LIN {X 0,Y 573.005,Z 611.639,A -85,B 0,C 180,E1 -2254.218,E2 -2254.218} C_VEL
LIN {X 0,Y 573.014,Z 607.193,A -85,B 0,C 180,E1 -2255.982,E2 -2255.982} C_VEL
LIN {X 0,Y 573.04,Z 602.476,A -85,B 0,C 180,E1 -2257.397,E2 -2257.397} C_VEL
LIN {X 0,Y 573.091,Z 594.867,A -85,B 0,C 180,E1 -2259.171,E2 -2259.171} C_VEL
LIN {X 0,Y 573.165,Z 587.276,A -85,B 0,C 180,E1 -2260.596,E2 -2260.596} C_VEL
LIN {X 0,Y 573.302,Z 578.228,A -85,B 0,C 180,E1 -2262.026,E2 -2262.026} C_VEL
LIN {X 0,Y 573.441,Z 567.442,A -85,B 0,C 180,E1 -2263.463,E2 -2263.463} C_VEL
LIN {X 0,Y 573.682,Z 556.314,A -85,B 0,C 180,E1 -2264.723,E2 -2264.723} C_VEL
LIN {X 0,Y 573.877,Z 544.168,A -85,B 0,C 180,E1 -2265.901,E2 -2265.901} C_VEL
LIN {X 0,Y 574.13,Z 530.904,A -85,B 0,C 180,E1 -2266.991,E2 -2266.991} C_VEL
LIN {X 0,Y 574.389,Z 517.891,A -85,B 0,C 180,E1 -2267.901,E2 -2267.901} C_VEL
LIN {X 0,Y 574.662,Z 504.072,A -85,B 0,C 180,E1 -2268.723,E2 -2268.723} C_VEL
LIN {X 0,Y 574.932,Z 489.306,A -85,B 0,C 180,E1 -2269.448,E2 -2269.448} C_VEL
LIN {X 0,Y 575.133,Z 474.014,A -85,B 0,C 180,E1 -2270.052,E2 -2270.052} C_VEL
LIN {X 0,Y 575.364,Z 457.285,A -85,B 0,C 180,E1 -2270.557,E2 -2270.557} C_VEL
LIN {X 0,Y 575.514,Z 441.109,A -85,B 0,C 180,E1 -2270.902,E2 -2270.902} C_VEL
LIN {X 0,Y 576.207,Z 242.353,A -85,B 0,C 180,E1 -2273.515,E2 -2273.515} C_VEL
LIN {X 0,Y 575.024,Z 234.784,A -85,B 0,C 180,E1 -2273.687,E2 -2273.687} C_VEL
LIN {X 0,Y 575.523,Z 201.562,A -85,B 0,C 180,E1 -2276.564,E2 -2276.564} C_VEL
LIN {X 0,Y 575.358,Z 193.757,A -85,B 0,C 180,E1 -2277.259,E2 -2277.259} C_VEL
LIN {X 0,Y 573.235,Z 186.394,A -85,B 0,C 180,E1 -2278.026,E2 -2278.026} C_VEL
LIN {X 0,Y 573.213,Z 186.396,A -85,B 0,C 180,E1 -2280.88,E2 -2280.88} C_VEL
LIN {X 0,Y 573.245,Z 186.393,A -85,B 0,C 180,E1 -2283.522,E2 -2283.522} C_VEL
LIN {X 0,Y 573.196,Z 186.394,A -85,B 0,C 180,E1 -2286.049,E2 -2286.049} C_VEL
LIN {X 0,Y 573.225,Z 186.392,A -85,B 0,C 180,E1 -2288.699,E2 -2288.699} C_VEL
LIN {X 0,Y 573.209,Z 186.396,A -85,B 0,C 180,E1 -2291.455,E2 -2291.455} C_VEL
LIN {X 0,Y 573.208,Z 186.391,A -85,B 0,C 180,E1 -2294.332,E2 -2294.332} C_VEL
LIN {X 0,Y 573.222,Z 186.395,A -85,B 0,C 180,E1 -2297.356,E2 -2297.356} C_VEL
LIN {X 0,Y 573.223,Z 186.389,A -85,B 0,C 180,E1 -2300.391,E2 -2300.391} C_VEL
LIN {X 0,Y 573.227,Z 186.396,A -85,B 0,C 180,E1 -2303.076,E2 -2303.076} C_VEL
LIN {X 0,Y 573.242,Z 186.388,A -85,B 0,C 180,E1 -2305.67,E2 -2305.67} C_VEL
LIN {X 0,Y 573.22,Z 186.387,A -85,B 0,C 180,E1 -2308.184,E2 -2308.184} C_VEL
LIN {X 0,Y 573.236,Z 186.392,A -85,B 0,C 180,E1 -2310.633,E2 -2310.633} C_VEL
LIN {X 0,Y 573.227,Z 186.394,A -85,B 0,C 180,E1 -2313.023,E2 -2313.023} C_VEL
LIN {X 0,Y 573.242,Z 186.39,A -85,B 0,C 180,E1 -2315.365,E2 -2315.365} C_VEL
LIN {X 0,Y 573.233,Z 186.388,A -85,B 0,C 180,E1 -2317.662,E2 -2317.662} C_VEL
LIN {X 0,Y 573.245,Z 186.39,A -85,B 0,C 180,E1 -2320.727,E2 -2320.727} C_VEL
LIN {X 0,Y 573.225,Z 186.389,A -85,B 0,C 180,E1 -2323.621,E2 -2323.621} C_VEL
LIN {X 0,Y 573.211,Z 186.394,A -85,B 0,C 180,E1 -2326.529,E2 -2326.529} C_VEL
LIN {X 0,Y 573.262,Z 186.384,A -85,B 0,C 180,E1 -2329.404,E2 -2329.404} C_VEL
LIN {X 0,Y 573.256,Z 186.387,A -85,B 0,C 180,E1 -2332.25,E2 -2332.25} C_VEL
LIN {X 0,Y 573.283,Z 186.381,A -85,B 0,C 180,E1 -2335.077,E2 -2335.077} C_VEL
LIN {X 0,Y 573.267,Z 186.38,A -85,B 0,C 180,E1 -2337.893,E2 -2337.893} C_VEL
LIN {X 0,Y 573.316,Z 186.387,A -85,B 0,C 180,E1 -2340.703,E2 -2340.703} C_VEL
LIN {X 0,Y 573.206,Z 186.389,A -85,B 0,C 180,E1 -2343.515,E2 -2343.515} C_VEL
LIN {X 0,Y 573.257,Z 186.382,A -85,B 0,C 180,E1 -2345.629,E2 -2345.629} C_VEL
LIN {X 0,Y 573.275,Z 186.39,A -85,B 0,C 180,E1 -2348.46,E2 -2348.46} C_VEL
LIN {X 0,Y 573.265,Z 186.381,A -85,B 0,C 180,E1 -2351.313,E2 -2351.313} C_VEL
LIN {X 0,Y 573.247,Z 186.393,A -85,B 0,C 180,E1 -2354.426,E2 -2354.426} C_VEL
LIN {X 0,Y 573.269,Z 186.383,A -85,B 0,C 180,E1 -2357.112,E2 -2357.112} C_VEL
LIN {X 0,Y 573.232,Z 186.388,A -85,B 0,C 180,E1 -2360.078,E2 -2360.078} C_VEL
LIN {X 0,Y 573.242,Z 186.387,A -85,B 0,C 180,E1 -2363.155,E2 -2363.155} C_VEL
LIN {X 0,Y 573.225,Z 186.391,A -85,B 0,C 180,E1 -2364.422,E2 -2364.422} C_VEL
LIN {X 0,Y 572.593,Z 186.472,A -85,B 0,C 180,E1 -2365.009,E2 -2365.009} C_VEL
LIN {X 0,Y 569.748,Z 186.824,A -85,B 0,C 180,E1 -2365.96,E2 -2365.96} C_VEL
LIN {X 0,Y 567.319,Z 187.128,A -85,B 0,C 180,E1 -2366.726,E2 -2366.726} C_VEL
LIN {X 0,Y 566.27,Z 187.254,A -85,B 0,C 180,E1 -2367.317,E2 -2367.317} C_VEL
LIN {X 0,Y 566.183,Z 187.264,A -85,B 0,C 180,E1 -2367.517,E2 -2367.517} C_VEL
LIN {X 0,Y 566.174,Z 187.268,A -85,B 0,C 180,E1 -2369.771,E2 -2369.771} C_VEL
LIN {X 0,Y 566.181,Z 187.271,A -85,B 0,C 180,E1 -2372.433,E2 -2372.433} C_VEL
LIN {X 0,Y 566.175,Z 187.268,A -85,B 0,C 180,E1 -2374.995,E2 -2374.995} C_VEL
LIN {X 0,Y 566.173,Z 187.267,A -85,B 0,C 180,E1 -2377.463,E2 -2377.463} C_VEL
LIN {X 0,Y 566.193,Z 187.27,A -85,B 0,C 180,E1 -2380.201,E2 -2380.201} C_VEL
LIN {X 0,Y 566.181,Z 187.266,A -85,B 0,C 180,E1 -2383.057,E2 -2383.057} C_VEL
LIN {X 0,Y 566.174,Z 187.271,A -85,B 0,C 180,E1 -2386.052,E2 -2386.052} C_VEL
LIN {X 0,Y 566.186,Z 187.265,A -85,B 0,C 180,E1 -2389.217,E2 -2389.217} C_VEL
LIN {X 0,Y 566.166,Z 187.269,A -85,B 0,C 180,E1 -2391.639,E2 -2391.639} C_VEL
LIN {X 0,Y 566.178,Z 187.271,A -85,B 0,C 180,E1 -2394.313,E2 -2394.313} C_VEL
LIN {X 0,Y 566.207,Z 187.263,A -85,B 0,C 180,E1 -2396.9,E2 -2396.9} C_VEL
LIN {X 0,Y 566.165,Z 187.269,A -85,B 0,C 180,E1 -2399.41,E2 -2399.41} C_VEL
LIN {X 0,Y 566.179,Z 187.273,A -85,B 0,C 180,E1 -2401.859,E2 -2401.859} C_VEL
LIN {X 0,Y 566.187,Z 187.271,A -85,B 0,C 180,E1 -2404.253,E2 -2404.253} C_VEL
LIN {X 0,Y 566.163,Z 187.269,A -85,B 0,C 180,E1 -2407.371,E2 -2407.371} C_VEL
LIN {X 0,Y 566.189,Z 187.271,A -85,B 0,C 180,E1 -2409.665,E2 -2409.665} C_VEL
LIN {X 0,Y 566.165,Z 187.277,A -85,B 0,C 180,E1 -2411.923,E2 -2411.923} C_VEL
LIN {X 0,Y 566.183,Z 187.267,A -85,B 0,C 180,E1 -2414.892,E2 -2414.892} C_VEL
LIN {X 0,Y 566.208,Z 187.272,A -85,B 0,C 180,E1 -2417.821,E2 -2417.821} C_VEL
LIN {X 0,Y 566.165,Z 187.276,A -85,B 0,C 180,E1 -2419.994,E2 -2419.994} C_VEL
LIN {X 0,Y 566.186,Z 187.267,A -85,B 0,C 180,E1 -2422.872,E2 -2422.872} C_VEL
LIN {X 0,Y 566.256,Z 187.256,A -85,B 0,C 180,E1 -2425.018,E2 -2425.018} C_VEL
LIN {X 0,Y 566.281,Z 187.263,A -85,B 0,C 180,E1 -2427.868,E2 -2427.868} C_VEL
LIN {X 0,Y 566.289,Z 187.262,A -85,B 0,C 180,E1 -2430.002,E2 -2430.002} C_VEL
LIN {X 0,Y 566.199,Z 187.414,A -85,B 0,C 180,E1 -2431.113,E2 -2431.113} C_VEL
LIN {X 0,Y 568.119,Z 194.679,A -85,B 0,C 180,E1 -2431.951,E2 -2431.951} C_VEL
LIN {X 0,Y 568.088,Z 205.896,A -85,B 0,C 180,E1 -2433.083,E2 -2433.083} C_VEL
LIN {X 0,Y 569.648,Z 213.911,A -85,B 0,C 180,E1 -2433.264,E2 -2433.264} C_VEL
LIN {X 0,Y 568.894,Z 411.449,A -85,B 0,C 180,E1 -2435.896,E2 -2435.896} C_VEL
LIN {X 0,Y 568.698,Z 428.048,A -85,B 0,C 180,E1 -2436.254,E2 -2436.254} C_VEL
LIN {X 0,Y 568.478,Z 444.08,A -85,B 0,C 180,E1 -2436.746,E2 -2436.746} C_VEL
LIN {X 0,Y 568.226,Z 458.901,A -85,B 0,C 180,E1 -2437.34,E2 -2437.34} C_VEL
LIN {X 0,Y 567.898,Z 474.039,A -85,B 0,C 180,E1 -2438.091,E2 -2438.091} C_VEL
LIN {X 0,Y 567.548,Z 489.027,A -85,B 0,C 180,E1 -2438.996,E2 -2438.996} C_VEL
LIN {X 0,Y 567.238,Z 502.812,A -85,B 0,C 180,E1 -2439.99,E2 -2439.99} C_VEL
LIN {X 0,Y 566.955,Z 515.623,A -85,B 0,C 180,E1 -2441.079,E2 -2441.079} C_VEL
LIN {X 0,Y 566.668,Z 528.371,A -85,B 0,C 180,E1 -2442.355,E2 -2442.355} C_VEL
LIN {X 0,Y 566.411,Z 539.253,A -85,B 0,C 180,E1 -2443.637,E2 -2443.637} C_VEL
LIN {X 0,Y 566.259,Z 548.723,A -85,B 0,C 180,E1 -2444.938,E2 -2444.938} C_VEL
LIN {X 0,Y 566.114,Z 557.804,A -85,B 0,C 180,E1 -2446.406,E2 -2446.406} C_VEL
LIN {X 0,Y 566.053,Z 564.614,A -85,B 0,C 180,E1 -2447.71,E2 -2447.71} C_VEL
LIN {X 0,Y 565.982,Z 571.522,A -85,B 0,C 180,E1 -2449.313,E2 -2449.313} C_VEL
LIN {X 0,Y 565.9,Z 576.436,A -85,B 0,C 180,E1 -2450.73,E2 -2450.73} C_VEL
LIN {X 0,Y 565.857,Z 579.615,A -85,B 0,C 180,E1 -2451.877,E2 -2451.877} C_VEL
LIN {X 0,Y 565.821,Z 582.884,A -85,B 0,C 180,E1 -2453.421,E2 -2453.421} C_VEL
LIN {X 0,Y 565.817,Z 584.97,A -85,B 0,C 180,E1 -2454.982,E2 -2454.982} C_VEL
LIN {X 0,Y 565.865,Z 585.906,A -85,B 0,C 180,E1 -2456.589,E2 -2456.589} C_VEL
LIN {X 0,Y 565.833,Z 585.679,A -85,B 0,C 180,E1 -2458.164,E2 -2458.164} C_VEL
LIN {X 0,Y 565.872,Z 584.221,A -85,B 0,C 180,E1 -2459.789,E2 -2459.789} C_VEL
LIN {X 0,Y 565.848,Z 581.384,A -85,B 0,C 180,E1 -2461.444,E2 -2461.444} C_VEL
LIN {X 0,Y 565.896,Z 577.134,A -85,B 0,C 180,E1 -2463.124,E2 -2463.124} C_VEL
LIN {X 0,Y 565.914,Z 572.939,A -85,B 0,C 180,E1 -2464.407,E2 -2464.407} C_VEL
LIN {X 0,Y 566.037,Z 566.63,A -85,B 0,C 180,E1 -2465.945,E2 -2465.945} C_VEL
LIN {X 0,Y 566.092,Z 558.995,A -85,B 0,C 180,E1 -2467.469,E2 -2467.469} C_VEL
LIN {X 0,Y 566.245,Z 550.521,A -85,B 0,C 180,E1 -2468.882,E2 -2468.882} C_VEL
LIN {X 0,Y 566.361,Z 541.331,A -85,B 0,C 180,E1 -2470.186,E2 -2470.186} C_VEL
LIN {X 0,Y 566.599,Z 529.811,A -85,B 0,C 180,E1 -2471.576,E2 -2471.576} C_VEL
LIN {X 0,Y 566.886,Z 518.399,A -85,B 0,C 180,E1 -2472.748,E2 -2472.748} C_VEL
LIN {X 0,Y 567.191,Z 504.81,A -85,B 0,C 180,E1 -2473.939,E2 -2473.939} C_VEL
LIN {X 0,Y 567.529,Z 490.173,A -85,B 0,C 180,E1 -2475.017,E2 -2475.017} C_VEL
LIN {X 0,Y 567.879,Z 476.319,A -85,B 0,C 180,E1 -2475.873,E2 -2475.873} C_VEL
LIN {X 0,Y 568.157,Z 461.078,A -85,B 0,C 180,E1 -2476.655,E2 -2476.655} C_VEL
LIN {X 0,Y 568.458,Z 445.107,A -85,B 0,C 180,E1 -2477.307,E2 -2477.307} C_VEL
LIN {X 0,Y 568.713,Z 429.222,A -85,B 0,C 180,E1 -2477.802,E2 -2477.802} C_VEL
LIN {X 0,Y 568.874,Z 412.275,A -85,B 0,C 180,E1 -2478.18,E2 -2478.18} C_VEL
LIN {X 0,Y 569.146,Z 352.079,A -85,B 0,C 180,E1 -2478.995,E2 -2478.995} C_VEL
LIN {X 0,Y 569.619,Z 213.402,A -85,B 0,C 180,E1 -2480.835,E2 -2480.835} C_VEL
LIN {X 0,Y 568.092,Z 205.827,A -85,B 0,C 180,E1 -2481.016,E2 -2481.016} C_VEL
LIN {X 0,Y 568.266,Z 195.751,A -85,B 0,C 180,E1 -2482.027,E2 -2482.027} C_VEL
LIN {X 0,Y 566.227,Z 187.267,A -85,B 0,C 180,E1 -2483.015,E2 -2483.015} C_VEL
LIN {X 0,Y 566.213,Z 187.271,A -85,B 0,C 180,E1 -2486.044,E2 -2486.044} C_VEL
LIN {X 0,Y 566.194,Z 187.271,A -85,B 0,C 180,E1 -2488.578,E2 -2488.578} C_VEL
LIN {X 0,Y 566.194,Z 187.266,A -85,B 0,C 180,E1 -2491.046,E2 -2491.046} C_VEL
LIN {X 0,Y 566.215,Z 187.264,A -85,B 0,C 180,E1 -2493.458,E2 -2493.458} C_VEL
LIN {X 0,Y 566.198,Z 187.271,A -85,B 0,C 180,E1 -2495.819,E2 -2495.819} C_VEL
LIN {X 0,Y 566.207,Z 187.263,A -85,B 0,C 180,E1 -2498.902,E2 -2498.902} C_VEL
LIN {X 0,Y 566.207,Z 187.264,A -85,B 0,C 180,E1 -2501.172,E2 -2501.172} C_VEL
LIN {X 0,Y 566.214,Z 187.263,A -85,B 0,C 180,E1 -2503.412,E2 -2503.412} C_VEL
LIN {X 0,Y 566.194,Z 187.268,A -85,B 0,C 180,E1 -2506.358,E2 -2506.358} C_VEL
LIN {X 0,Y 566.232,Z 187.26,A -85,B 0,C 180,E1 -2508.675,E2 -2508.675} C_VEL
LIN {X 0,Y 566.224,Z 187.265,A -85,B 0,C 180,E1 -2511.434,E2 -2511.434} C_VEL
LIN {X 0,Y 566.251,Z 187.26,A -85,B 0,C 180,E1 -2514.301,E2 -2514.301} C_VEL
LIN {X 0,Y 566.272,Z 187.263,A -85,B 0,C 180,E1 -2517.866,E2 -2517.866} C_VEL
LIN {X 0,Y 566.296,Z 187.252,A -85,B 0,C 180,E1 -2520.711,E2 -2520.711} C_VEL
LIN {X 0,Y 566.265,Z 187.256,A -85,B 0,C 180,E1 -2522.845,E2 -2522.845} C_VEL
LIN {X 0,Y 566.253,Z 187.266,A -85,B 0,C 180,E1 -2525.698,E2 -2525.698} C_VEL
LIN {X 0,Y 566.2,Z 187.264,A -85,B 0,C 180,E1 -2528.566,E2 -2528.566} C_VEL
LIN {X 0,Y 566.238,Z 187.267,A -85,B 0,C 180,E1 -2531.454,E2 -2531.454} C_VEL
LIN {X 0,Y 566.225,Z 187.261,A -85,B 0,C 180,E1 -2534.504,E2 -2534.504} C_VEL
LIN {X 0,Y 566.194,Z 187.273,A -85,B 0,C 180,E1 -2537.331,E2 -2537.331} C_VEL
LIN {X 0,Y 566.202,Z 187.264,A -85,B 0,C 180,E1 -2540.337,E2 -2540.337} C_VEL
LIN {X 0,Y 566.167,Z 187.277,A -85,B 0,C 180,E1 -2543.281,E2 -2543.281} C_VEL
LIN {X 0,Y 566.204,Z 187.266,A -85,B 0,C 180,E1 -2545.749,E2 -2545.749} C_VEL
LIN {X 0,Y 566.2,Z 187.264,A -85,B 0,C 180,E1 -2548.202,E2 -2548.202} C_VEL
LIN {X 0,Y 566.185,Z 187.274,A -85,B 0,C 180,E1 -2551.076,E2 -2551.076} C_VEL
LIN {X 0,Y 566.195,Z 187.266,A -85,B 0,C 180,E1 -2553.732,E2 -2553.732} C_VEL
LIN {X 0,Y 566.197,Z 187.266,A -85,B 0,C 180,E1 -2556.57,E2 -2556.57} C_VEL
LIN {X 0,Y 566.21,Z 187.264,A -85,B 0,C 180,E1 -2559.685,E2 -2559.685} C_VEL
LIN {X 0,Y 566.192,Z 187.273,A -85,B 0,C 180,E1 -2562.916,E2 -2562.916} C_VEL
LIN {X 0,Y 566.192,Z 187.266,A -85,B 0,C 180,E1 -2566.049,E2 -2566.049} C_VEL
LIN {X 0,Y 566.201,Z 187.269,A -85,B 0,C 180,E1 -2569.214,E2 -2569.214} C_VEL
LIN {X 0,Y 566.182,Z 187.268,A -85,B 0,C 180,E1 -2571.636,E2 -2571.636} C_VEL
LIN {X 0,Y 566.149,Z 187.274,A -85,B 0,C 180,E1 -2574.306,E2 -2574.306} C_VEL
LIN {X 0,Y 566.207,Z 187.272,A -85,B 0,C 180,E1 -2576.896,E2 -2576.896} C_VEL
LIN {X 0,Y 566.169,Z 187.272,A -85,B 0,C 180,E1 -2579.406,E2 -2579.406} C_VEL
LIN {X 0,Y 566.199,Z 187.403,A -85,B 0,C 180,E1 -2581.72,E2 -2581.72} C_VEL
LIN {X 0,Y 568.874,Z 196.818,A -85,B 0,C 180,E1 -2582.699,E2 -2582.699} C_VEL
LIN {X 0,Y 568.459,Z 225.836,A -85,B 0,C 180,E1 -2585.24,E2 -2585.24} C_VEL
LIN {X 0,Y 568.336,Z 234.981,A -85,B 0,C 180,E1 -2586.035,E2 -2586.035} C_VEL
LIN {X 0,Y 569.689,Z 242.719,A -85,B 0,C 180,E1 -2586.204,E2 -2586.204} C_VEL
LIN {X 0,Y 568.891,Z 442.37,A -85,B 0,C 180,E1 -2588.863,E2 -2588.863} C_VEL
LIN {X 0,Y 568.704,Z 458.969,A -85,B 0,C 180,E1 -2589.235,E2 -2589.235} C_VEL
LIN {X 0,Y 568.407,Z 475.212,A -85,B 0,C 180,E1 -2589.744,E2 -2589.744} C_VEL
LIN {X 0,Y 568.148,Z 491.363,A -85,B 0,C 180,E1 -2590.407,E2 -2590.407} C_VEL
LIN {X 0,Y 567.88,Z 505.696,A -85,B 0,C 180,E1 -2591.135,E2 -2591.135} C_VEL
LIN {X 0,Y 567.526,Z 520.754,A -85,B 0,C 180,E1 -2592.064,E2 -2592.064} C_VEL
LIN {X 0,Y 567.172,Z 534.373,A -85,B 0,C 180,E1 -2593.069,E2 -2593.069} C_VEL
LIN {X 0,Y 566.917,Z 547.056,A -85,B 0,C 180,E1 -2594.172,E2 -2594.172} C_VEL
LIN {X 0,Y 566.626,Z 558.635,A -85,B 0,C 180,E1 -2595.341,E2 -2595.341} C_VEL
LIN {X 0,Y 566.435,Z 570.328,A -85,B 0,C 180,E1 -2596.729,E2 -2596.729} C_VEL
LIN {X 0,Y 566.24,Z 580.663,A -85,B 0,C 180,E1 -2598.181,E2 -2598.181} C_VEL
LIN {X 0,Y 566.12,Z 589.276,A -85,B 0,C 180,E1 -2599.628,E2 -2599.628} C_VEL
LIN {X 0,Y 566.002,Z 596.483,A -85,B 0,C 180,E1 -2601.07,E2 -2601.07} C_VEL
LIN {X 0,Y 565.969,Z 602.461,A -85,B 0,C 180,E1 -2602.507,E2 -2602.507} C_VEL
LIN {X 0,Y 565.916,Z 607.182,A -85,B 0,C 180,E1 -2603.939,E2 -2603.939} C_VEL
LIN {X 0,Y 565.911,Z 611.633,A -85,B 0,C 180,E1 -2605.725,E2 -2605.725} C_VEL
LIN {X 0,Y 565.866,Z 614.087,A -85,B 0,C 180,E1 -2607.151,E2 -2607.151} C_VEL
LIN {X 0,Y 565.839,Z 615.479,A -85,B 0,C 180,E1 -2608.575,E2 -2608.575} C_VEL
LIN {X 0,Y 565.834,Z 616,A -85,B 0,C 180,E1 -2609.998,E2 -2609.998} C_VEL
LIN {X 0,Y 565.839,Z 615.481,A -85,B 0,C 180,E1 -2611.422,E2 -2611.422} C_VEL
LIN {X 0,Y 565.865,Z 614.091,A -85,B 0,C 180,E1 -2612.846,E2 -2612.846} C_VEL
LIN {X 0,Y 565.91,Z 611.64,A -85,B 0,C 180,E1 -2614.271,E2 -2614.271} C_VEL
LIN {X 0,Y 565.914,Z 607.194,A -85,B 0,C 180,E1 -2616.057,E2 -2616.057} C_VEL
LIN {X 0,Y 565.968,Z 602.475,A -85,B 0,C 180,E1 -2617.49,E2 -2617.49} C_VEL
LIN {X 0,Y 566.009,Z 596.499,A -85,B 0,C 180,E1 -2618.927,E2 -2618.927} C_VEL
LIN {X 0,Y 566.126,Z 588.289,A -85,B 0,C 180,E1 -2620.549,E2 -2620.549} C_VEL
LIN {X 0,Y 566.243,Z 579.457,A -85,B 0,C 180,E1 -2621.997,E2 -2621.997} C_VEL
LIN {X 0,Y 566.425,Z 568.926,A -85,B 0,C 180,E1 -2623.45,E2 -2623.45} C_VEL
LIN {X 0,Y 566.682,Z 557.62,A -85,B 0,C 180,E1 -2624.772,E2 -2624.772} C_VEL
LIN {X 0,Y 566.931,Z 545.143,A -85,B 0,C 180,E1 -2626.009,E2 -2626.009} C_VEL
LIN {X 0,Y 567.231,Z 532.075,A -85,B 0,C 180,E1 -2627.111,E2 -2627.111} C_VEL
LIN {X 0,Y 567.58,Z 517.887,A -85,B 0,C 180,E1 -2628.123,E2 -2628.123} C_VEL
LIN {X 0,Y 567.898,Z 504.075,A -85,B 0,C 180,E1 -2628.954,E2 -2628.954} C_VEL
LIN {X 0,Y 568.221,Z 488.328,A -85,B 0,C 180,E1 -2629.733,E2 -2629.733} C_VEL
LIN {X 0,Y 568.522,Z 471.414,A -85,B 0,C 180,E1 -2630.39,E2 -2630.39} C_VEL
LIN {X 0,Y 568.744,Z 455.452,A -85,B 0,C 180,E1 -2630.854,E2 -2630.854} C_VEL
LIN {X 0,Y 568.909,Z 439.603,A -85,B 0,C 180,E1 -2631.18,E2 -2631.18} C_VEL
LIN {X 0,Y 569.711,Z 243.13,A -85,B 0,C 180,E1 -2633.789,E2 -2633.789} C_VEL
LIN {X 0,Y 568.349,Z 234.863,A -85,B 0,C 180,E1 -2633.975,E2 -2633.975} C_VEL
LIN {X 0,Y 568.919,Z 199.873,A -85,B 0,C 180,E1 -2637.032,E2 -2637.032} C_VEL
LIN {X 0,Y 568.647,Z 195.805,A -85,B 0,C 180,E1 -2637.408,E2 -2637.408} C_VEL
LIN {X 0,Y 566.193,Z 187.272,A -85,B 0,C 180,E1 -2638.322,E2 -2638.322} C_VEL
LIN {X 0,Y 566.176,Z 187.274,A -85,B 0,C 180,E1 -2641.074,E2 -2641.074} C_VEL
LIN {X 0,Y 566.194,Z 187.269,A -85,B 0,C 180,E1 -2643.732,E2 -2643.732} C_VEL
LIN {X 0,Y 566.18,Z 187.269,A -85,B 0,C 180,E1 -2646.568,E2 -2646.568} C_VEL
LIN {X 0,Y 566.19,Z 187.267,A -85,B 0,C 180,E1 -2649.683,E2 -2649.683} C_VEL
LIN {X 0,Y 566.168,Z 187.268,A -85,B 0,C 180,E1 -2652.087,E2 -2652.087} C_VEL
LIN {X 0,Y 566.149,Z 187.279,A -85,B 0,C 180,E1 -2655.034,E2 -2655.034} C_VEL
LIN {X 0,Y 566.19,Z 187.266,A -85,B 0,C 180,E1 -2657.911,E2 -2657.911} C_VEL
LIN {X 0,Y 566.197,Z 187.268,A -85,B 0,C 180,E1 -2660.725,E2 -2660.725} C_VEL
LIN {X 0,Y 566.188,Z 187.265,A -85,B 0,C 180,E1 -2663.782,E2 -2663.782} C_VEL
LIN {X 0,Y 566.182,Z 187.267,A -85,B 0,C 180,E1 -2666.264,E2 -2666.264} C_VEL
LIN {X 0,Y 566.17,Z 187.273,A -85,B 0,C 180,E1 -2668.92,E2 -2668.92} C_VEL
LIN {X 0,Y 566.197,Z 187.264,A -85,B 0,C 180,E1 -2671.857,E2 -2671.857} C_VEL
LIN {X 0,Y 566.182,Z 187.263,A -85,B 0,C 180,E1 -2674.25,E2 -2674.25} C_VEL
LIN {X 0,Y 566.192,Z 187.268,A -85,B 0,C 180,E1 -2677.369,E2 -2677.369} C_VEL
LIN {X 0,Y 566.182,Z 187.265,A -85,B 0,C 180,E1 -2680.419,E2 -2680.419} C_VEL
LIN {X 0,Y 566.188,Z 187.267,A -85,B 0,C 180,E1 -2683.412,E2 -2683.412} C_VEL
LIN {X 0,Y 566.172,Z 187.268,A -85,B 0,C 180,E1 -2686.359,E2 -2686.359} C_VEL
LIN {X 0,Y 566.24,Z 187.26,A -85,B 0,C 180,E1 -2689.271,E2 -2689.271} C_VEL
LIN {X 0,Y 566.208,Z 187.264,A -85,B 0,C 180,E1 -2692.153,E2 -2692.153} C_VEL
LIN {X 0,Y 566.255,Z 187.257,A -85,B 0,C 180,E1 -2695.016,E2 -2695.016} C_VEL
LIN {X 0,Y 566.239,Z 187.255,A -85,B 0,C 180,E1 -2697.866,E2 -2697.866} C_VEL
LIN {X 0,Y 566.284,Z 187.263,A -85,B 0,C 180,E1 -2700.711,E2 -2700.711} C_VEL
LIN {X 0,Y 566.158,Z 187.267,A -85,B 0,C 180,E1 -2703.559,E2 -2703.559} C_VEL
LIN {X 0,Y 566.225,Z 187.258,A -85,B 0,C 180,E1 -2705.699,E2 -2705.699} C_VEL
LIN {X 0,Y 566.217,Z 187.271,A -85,B 0,C 180,E1 -2708.566,E2 -2708.566} C_VEL
LIN {X 0,Y 566.217,Z 187.257,A -85,B 0,C 180,E1 -2711.455,E2 -2711.455} C_VEL
LIN {X 0,Y 566.2,Z 187.272,A -85,B 0,C 180,E1 -2714.508,E2 -2714.508} C_VEL
LIN {X 0,Y 566.198,Z 187.262,A -85,B 0,C 180,E1 -2717.332,E2 -2717.332} C_VEL
LIN {X 0,Y 566.195,Z 187.269,A -85,B 0,C 180,E1 -2720.338,E2 -2720.338} C_VEL
LIN {X 0,Y 566.2,Z 187.263,A -85,B 0,C 180,E1 -2723.404,E2 -2723.404} C_VEL
LIN {X 0,Y 566.183,Z 187.264,A -85,B 0,C 180,E1 -2725.751,E2 -2725.751} C_VEL
LIN {X 0,Y 566.183,Z 187.264,A -85,B 0,C 180,E1 -2727.517,E2 -2727.517} C_VEL
LIN {X 0,Y 565.508,Z 187.355,A -85,B 0,C 180,E1 -2728.111,E2 -2728.111} C_VEL
LIN {X 0,Y 562.638,Z 187.712,A -85,B 0,C 180,E1 -2729.074,E2 -2729.074} C_VEL
LIN {X 0,Y 560.221,Z 188.013,A -85,B 0,C 180,E1 -2729.85,E2 -2729.85} C_VEL
LIN {X 0,Y 559.192,Z 188.144,A -85,B 0,C 180,E1 -2730.449,E2 -2730.449} C_VEL
LIN {X 0,Y 559.112,Z 188.148,A -85,B 0,C 180,E1 -2730.651,E2 -2730.651} C_VEL
LIN {X 0,Y 559.133,Z 188.141,A -85,B 0,C 180,E1 -2733.577,E2 -2733.577} C_VEL
LIN {X 0,Y 559.137,Z 188.151,A -85,B 0,C 180,E1 -2736.45,E2 -2736.45} C_VEL
LIN {X 0,Y 559.15,Z 188.139,A -85,B 0,C 180,E1 -2738.937,E2 -2738.937} C_VEL
LIN {X 0,Y 559.166,Z 188.142,A -85,B 0,C 180,E1 -2741.771,E2 -2741.771} C_VEL
LIN {X 0,Y 559.115,Z 188.145,A -85,B 0,C 180,E1 -2744.742,E2 -2744.742} C_VEL
LIN {X 0,Y 559.134,Z 188.144,A -85,B 0,C 180,E1 -2747.258,E2 -2747.258} C_VEL
LIN {X 0,Y 559.162,Z 188.147,A -85,B 0,C 180,E1 -2750.137,E2 -2750.137} C_VEL
LIN {X 0,Y 559.128,Z 188.145,A -85,B 0,C 180,E1 -2752.894,E2 -2752.894} C_VEL
LIN {X 0,Y 559.153,Z 188.148,A -85,B 0,C 180,E1 -2756.054,E2 -2756.054} C_VEL
LIN {X 0,Y 559.141,Z 188.143,A -85,B 0,C 180,E1 -2758.983,E2 -2758.983} C_VEL
LIN {X 0,Y 559.125,Z 188.148,A -85,B 0,C 180,E1 -2761.628,E2 -2761.628} C_VEL
LIN {X 0,Y 559.153,Z 188.149,A -85,B 0,C 180,E1 -2763.905,E2 -2763.905} C_VEL
LIN {X 0,Y 559.109,Z 188.147,A -85,B 0,C 180,E1 -2767.069,E2 -2767.069} C_VEL
LIN {X 0,Y 559.158,Z 188.143,A -85,B 0,C 180,E1 -2769.397,E2 -2769.397} C_VEL
LIN {X 0,Y 559.116,Z 188.151,A -85,B 0,C 180,E1 -2771.687,E2 -2771.687} C_VEL
LIN {X 0,Y 559.131,Z 188.146,A -85,B 0,C 180,E1 -2774.697,E2 -2774.697} C_VEL
LIN {X 0,Y 559.167,Z 188.147,A -85,B 0,C 180,E1 -2777.665,E2 -2777.665} C_VEL
LIN {X 0,Y 559.127,Z 188.154,A -85,B 0,C 180,E1 -2779.867,E2 -2779.867} C_VEL
LIN {X 0,Y 559.144,Z 188.151,A -85,B 0,C 180,E1 -2782.055,E2 -2782.055} C_VEL
LIN {X 0,Y 559.232,Z 188.131,A -85,B 0,C 180,E1 -2784.955,E2 -2784.955} C_VEL
LIN {X 0,Y 559.251,Z 188.138,A -85,B 0,C 180,E1 -2787.841,E2 -2787.841} C_VEL
LIN {X 0,Y 559.257,Z 188.138,A -85,B 0,C 180,E1 -2790.002,E2 -2790.002} C_VEL
LIN {X 0,Y 559.139,Z 188.286,A -85,B 0,C 180,E1 -2790.834,E2 -2790.834} C_VEL
LIN {X 0,Y 561.367,Z 196.459,A -85,B 0,C 180,E1 -2791.795,E2 -2791.795} C_VEL
LIN {X 0,Y 561.384,Z 206.119,A -85,B 0,C 180,E1 -2792.782,E2 -2792.782} C_VEL
LIN {X 0,Y 563.166,Z 215.478,A -85,B 0,C 180,E1 -2792.993,E2 -2792.993} C_VEL
LIN {X 0,Y 562.281,Z 411.044,A -85,B 0,C 180,E1 -2795.628,E2 -2795.628} C_VEL
LIN {X 0,Y 562.061,Z 427.8,A -85,B 0,C 180,E1 -2795.99,E2 -2795.99} C_VEL
LIN {X 0,Y 561.792,Z 444.567,A -85,B 0,C 180,E1 -2796.511,E2 -2796.511} C_VEL
LIN {X 0,Y 561.488,Z 460.073,A -85,B 0,C 180,E1 -2797.147,E2 -2797.147} C_VEL
LIN {X 0,Y 561.095,Z 475.245,A -85,B 0,C 180,E1 -2797.921,E2 -2797.921} C_VEL
LIN {X 0,Y 560.706,Z 489.983,A -85,B 0,C 180,E1 -2798.834,E2 -2798.834} C_VEL
LIN {X 0,Y 560.303,Z 504.755,A -85,B 0,C 180,E1 -2799.933,E2 -2799.933} C_VEL
LIN {X 0,Y 559.998,Z 517.284,A -85,B 0,C 180,E1 -2801.035,E2 -2801.035} C_VEL
LIN {X 0,Y 559.656,Z 529.795,A -85,B 0,C 180,E1 -2802.328,E2 -2802.328} C_VEL
LIN {X 0,Y 559.41,Z 540.503,A -85,B 0,C 180,E1 -2803.626,E2 -2803.626} C_VEL
LIN {X 0,Y 559.222,Z 550.788,A -85,B 0,C 180,E1 -2805.099,E2 -2805.099} C_VEL
LIN {X 0,Y 559.028,Z 559.71,A -85,B 0,C 180,E1 -2806.62,E2 -2806.62} C_VEL
LIN {X 0,Y 558.963,Z 566.24,A -85,B 0,C 180,E1 -2807.943,E2 -2807.943} C_VEL
LIN {X 0,Y 558.909,Z 572.318,A -85,B 0,C 180,E1 -2809.422,E2 -2809.422} C_VEL
LIN {X 0,Y 558.835,Z 577.469,A -85,B 0,C 180,E1 -2811.004,E2 -2811.004} C_VEL
LIN {X 0,Y 558.759,Z 580.485,A -85,B 0,C 180,E1 -2812.17,E2 -2812.17} C_VEL
LIN {X 0,Y 558.714,Z 583.438,A -85,B 0,C 180,E1 -2813.737,E2 -2813.737} C_VEL
LIN {X 0,Y 558.729,Z 585.293,A -85,B 0,C 180,E1 -2815.321,E2 -2815.321} C_VEL
LIN {X 0,Y 558.753,Z 585.98,A -85,B 0,C 180,E1 -2816.925,E2 -2816.925} C_VEL
LIN {X 0,Y 558.733,Z 585.434,A -85,B 0,C 180,E1 -2818.554,E2 -2818.554} C_VEL
LIN {X 0,Y 558.787,Z 583.664,A -85,B 0,C 180,E1 -2820.205,E2 -2820.205} C_VEL
LIN {X 0,Y 558.765,Z 580.561,A -85,B 0,C 180,E1 -2821.889,E2 -2821.889} C_VEL
LIN {X 0,Y 558.833,Z 575.974,A -85,B 0,C 180,E1 -2823.598,E2 -2823.598} C_VEL
LIN {X 0,Y 558.914,Z 569.714,A -85,B 0,C 180,E1 -2825.34,E2 -2825.34} C_VEL
LIN {X 0,Y 559.014,Z 563.441,A -85,B 0,C 180,E1 -2826.739,E2 -2826.739} C_VEL
LIN {X 0,Y 559.127,Z 555.529,A -85,B 0,C 180,E1 -2828.217,E2 -2828.217} C_VEL
LIN {X 0,Y 559.28,Z 546.601,A -85,B 0,C 180,E1 -2829.623,E2 -2829.623} C_VEL
LIN {X 0,Y 559.553,Z 535.49,A -85,B 0,C 180,E1 -2831.096,E2 -2831.096} C_VEL
LIN {X 0,Y 559.834,Z 524.122,A -85,B 0,C 180,E1 -2832.374,E2 -2832.374} C_VEL
LIN {X 0,Y 560.147,Z 510.927,A -85,B 0,C 180,E1 -2833.636,E2 -2833.636} C_VEL
LIN {X 0,Y 560.544,Z 497.461,A -85,B 0,C 180,E1 -2834.724,E2 -2834.724} C_VEL
LIN {X 0,Y 560.878,Z 483.034,A -85,B 0,C 180,E1 -2835.709,E2 -2835.709} C_VEL
LIN {X 0,Y 561.288,Z 467.761,A -85,B 0,C 180,E1 -2836.571,E2 -2836.571} C_VEL
LIN {X 0,Y 561.637,Z 452.941,A -85,B 0,C 180,E1 -2837.255,E2 -2837.255} C_VEL
LIN {X 0,Y 561.917,Z 436.364,A -85,B 0,C 180,E1 -2837.854,E2 -2837.854} C_VEL
LIN {X 0,Y 562.187,Z 419.827,A -85,B 0,C 180,E1 -2838.29,E2 -2838.29} C_VEL
LIN {X 0,Y 562.362,Z 402.663,A -85,B 0,C 180,E1 -2838.592,E2 -2838.592} C_VEL
LIN {X 0,Y 563.18,Z 215.299,A -85,B 0,C 180,E1 -2841.098,E2 -2841.098} C_VEL
LIN {X 0,Y 561.398,Z 206.025,A -85,B 0,C 180,E1 -2841.32,E2 -2841.32} C_VEL
LIN {X 0,Y 561.57,Z 197.606,A -85,B 0,C 180,E1 -2842.176,E2 -2842.176} C_VEL
LIN {X 0,Y 559.168,Z 188.146,A -85,B 0,C 180,E1 -2843.304,E2 -2843.304} C_VEL
LIN {X 0,Y 559.165,Z 188.148,A -85,B 0,C 180,E1 -2846.425,E2 -2846.425} C_VEL
LIN {X 0,Y 559.155,Z 188.144,A -85,B 0,C 180,E1 -2848.98,E2 -2848.98} C_VEL
LIN {X 0,Y 559.169,Z 188.143,A -85,B 0,C 180,E1 -2851.618,E2 -2851.618} C_VEL
LIN {X 0,Y 559.18,Z 188.145,A -85,B 0,C 180,E1 -2853.902,E2 -2853.902} C_VEL
LIN {X 0,Y 559.142,Z 188.147,A -85,B 0,C 180,E1 -2856.57,E2 -2856.57} C_VEL
LIN {X 0,Y 559.178,Z 188.139,A -85,B 0,C 180,E1 -2859.395,E2 -2859.395} C_VEL
LIN {X 0,Y 559.149,Z 188.148,A -85,B 0,C 180,E1 -2861.685,E2 -2861.685} C_VEL
LIN {X 0,Y 559.165,Z 188.149,A -85,B 0,C 180,E1 -2863.947,E2 -2863.947} C_VEL
LIN {X 0,Y 559.169,Z 188.146,A -85,B 0,C 180,E1 -2866.184,E2 -2866.184} C_VEL
LIN {X 0,Y 559.192,Z 188.138,A -85,B 0,C 180,E1 -2869.133,E2 -2869.133} C_VEL
LIN {X 0,Y 559.2,Z 188.143,A -85,B 0,C 180,E1 -2872.053,E2 -2872.053} C_VEL
LIN {X 0,Y 559.249,Z 188.13,A -85,B 0,C 180,E1 -2874.953,E2 -2874.953} C_VEL
LIN {X 0,Y 559.244,Z 188.138,A -85,B 0,C 180,E1 -2877.839,E2 -2877.839} C_VEL
LIN {X 0,Y 559.267,Z 188.128,A -85,B 0,C 180,E1 -2880.72,E2 -2880.72} C_VEL
LIN {X 0,Y 559.233,Z 188.132,A -85,B 0,C 180,E1 -2882.881,E2 -2882.881} C_VEL
LIN {X 0,Y 559.222,Z 188.141,A -85,B 0,C 180,E1 -2885.77,E2 -2885.77} C_VEL
LIN {X 0,Y 559.165,Z 188.141,A -85,B 0,C 180,E1 -2888.674,E2 -2888.674} C_VEL
LIN {X 0,Y 559.201,Z 188.144,A -85,B 0,C 180,E1 -2891.6,E2 -2891.6} C_VEL
LIN {X 0,Y 559.197,Z 188.137,A -85,B 0,C 180,E1 -2894.595,E2 -2894.595} C_VEL
LIN {X 0,Y 559.137,Z 188.151,A -85,B 0,C 180,E1 -2897.557,E2 -2897.557} C_VEL
LIN {X 0,Y 559.161,Z 188.144,A -85,B 0,C 180,E1 -2899.837,E2 -2899.837} C_VEL
LIN {X 0,Y 559.136,Z 188.144,A -85,B 0,C 180,E1 -2902.153,E2 -2902.153} C_VEL
LIN {X 0,Y 559.172,Z 188.148,A -85,B 0,C 180,E1 -2905.298,E2 -2905.298} C_VEL
LIN {X 0,Y 559.154,Z 188.145,A -85,B 0,C 180,E1 -2907.713,E2 -2907.713} C_VEL
LIN {X 0,Y 559.146,Z 188.143,A -85,B 0,C 180,E1 -2910.183,E2 -2910.183} C_VEL
LIN {X 0,Y 559.15,Z 188.145,A -85,B 0,C 180,E1 -2912.715,E2 -2912.715} C_VEL
LIN {X 0,Y 559.124,Z 188.152,A -85,B 0,C 180,E1 -2915.324,E2 -2915.324} C_VEL
LIN {X 0,Y 559.128,Z 188.145,A -85,B 0,C 180,E1 -2918.018,E2 -2918.018} C_VEL
LIN {X 0,Y 559.153,Z 188.148,A -85,B 0,C 180,E1 -2920.812,E2 -2920.812} C_VEL
LIN {X 0,Y 559.109,Z 188.148,A -85,B 0,C 180,E1 -2923.737,E2 -2923.737} C_VEL
LIN {X 0,Y 559.134,Z 188.147,A -85,B 0,C 180,E1 -2926.265,E2 -2926.265} C_VEL
LIN {X 0,Y 559.153,Z 188.148,A -85,B 0,C 180,E1 -2929.187,E2 -2929.187} C_VEL
LIN {X 0,Y 559.129,Z 188.146,A -85,B 0,C 180,E1 -2931.982,E2 -2931.982} C_VEL
LIN {X 0,Y 559.128,Z 188.153,A -85,B 0,C 180,E1 -2934.787,E2 -2934.787} C_VEL
LIN {X 0,Y 559.15,Z 188.145,A -85,B 0,C 180,E1 -2937.365,E2 -2937.365} C_VEL
LIN {X 0,Y 559.12,Z 188.151,A -85,B 0,C 180,E1 -2940.147,E2 -2940.147} C_VEL
LIN {X 0,Y 559.154,Z 188.273,A -85,B 0,C 180,E1 -2941.431,E2 -2941.431} C_VEL
LIN {X 0,Y 562.231,Z 198.956,A -85,B 0,C 180,E1 -2942.562,E2 -2942.562} C_VEL
LIN {X 0,Y 561.683,Z 230.083,A -85,B 0,C 180,E1 -2945.316,E2 -2945.316} C_VEL
LIN {X 0,Y 561.666,Z 235.278,A -85,B 0,C 180,E1 -2945.744,E2 -2945.744} C_VEL
LIN {X 0,Y 563.206,Z 244.105,A -85,B 0,C 180,E1 -2945.935,E2 -2945.935} C_VEL
LIN {X 0,Y 562.257,Z 440.874,A -85,B 0,C 180,E1 -2948.578,E2 -2948.578} C_VEL
LIN {X 0,Y 562.074,Z 457.137,A -85,B 0,C 180,E1 -2948.931,E2 -2948.931} C_VEL
LIN {X 0,Y 561.784,Z 473.911,A -85,B 0,C 180,E1 -2949.446,E2 -2949.446} C_VEL
LIN {X 0,Y 561.495,Z 489.98,A -85,B 0,C 180,E1 -2950.099,E2 -2950.099} C_VEL
LIN {X 0,Y 561.137,Z 504.017,A -85,B 0,C 180,E1 -2950.805,E2 -2950.805} C_VEL
LIN {X 0,Y 560.741,Z 519.256,A -85,B 0,C 180,E1 -2951.739,E2 -2951.739} C_VEL
LIN {X 0,Y 560.35,Z 533.2,A -85,B 0,C 180,E1 -2952.763,E2 -2952.763} C_VEL
LIN {X 0,Y 559.999,Z 547.055,A -85,B 0,C 180,E1 -2953.971,E2 -2953.971} C_VEL
LIN {X 0,Y 559.658,Z 559.256,A -85,B 0,C 180,E1 -2955.225,E2 -2955.225} C_VEL
LIN {X 0,Y 559.43,Z 570.329,A -85,B 0,C 180,E1 -2956.56,E2 -2956.56} C_VEL
LIN {X 0,Y 559.221,Z 580.662,A -85,B 0,C 180,E1 -2958.031,E2 -2958.031} C_VEL
LIN {X 0,Y 559.074,Z 589.276,A -85,B 0,C 180,E1 -2959.496,E2 -2959.496} C_VEL
LIN {X 0,Y 558.938,Z 596.484,A -85,B 0,C 180,E1 -2960.956,E2 -2960.956} C_VEL
LIN {X 0,Y 558.895,Z 602.46,A -85,B 0,C 180,E1 -2962.411,E2 -2962.411} C_VEL
LIN {X 0,Y 558.864,Z 608.244,A -85,B 0,C 180,E1 -2964.225,E2 -2964.225} C_VEL
LIN {X 0,Y 558.805,Z 611.633,A -85,B 0,C 180,E1 -2965.671,E2 -2965.671} C_VEL
LIN {X 0,Y 558.787,Z 614.087,A -85,B 0,C 180,E1 -2967.115,E2 -2967.115} C_VEL
LIN {X 0,Y 558.739,Z 615.478,A -85,B 0,C 180,E1 -2968.557,E2 -2968.557} C_VEL
LIN {X 0,Y 558.735,Z 616,A -85,B 0,C 180,E1 -2969.998,E2 -2969.998} C_VEL
LIN {X 0,Y 558.739,Z 615.48,A -85,B 0,C 180,E1 -2971.44,E2 -2971.44} C_VEL
LIN {X 0,Y 558.787,Z 614.091,A -85,B 0,C 180,E1 -2972.882,E2 -2972.882} C_VEL
LIN {X 0,Y 558.805,Z 611.639,A -85,B 0,C 180,E1 -2974.326,E2 -2974.326} C_VEL
LIN {X 0,Y 558.863,Z 608.256,A -85,B 0,C 180,E1 -2975.772,E2 -2975.772} C_VEL
LIN {X 0,Y 558.893,Z 602.475,A -85,B 0,C 180,E1 -2977.585,E2 -2977.585} C_VEL
LIN {X 0,Y 558.945,Z 596.5,A -85,B 0,C 180,E1 -2979.041,E2 -2979.041} C_VEL
LIN {X 0,Y 559.072,Z 589.295,A -85,B 0,C 180,E1 -2980.5,E2 -2980.5} C_VEL
LIN {X 0,Y 559.216,Z 580.686,A -85,B 0,C 180,E1 -2981.966,E2 -2981.966} C_VEL
LIN {X 0,Y 559.428,Z 570.356,A -85,B 0,C 180,E1 -2983.437,E2 -2983.437} C_VEL
LIN {X 0,Y 559.652,Z 559.278,A -85,B 0,C 180,E1 -2984.772,E2 -2984.772} C_VEL
LIN {X 0,Y 559.982,Z 547.091,A -85,B 0,C 180,E1 -2986.026,E2 -2986.026} C_VEL
LIN {X 0,Y 560.338,Z 533.245,A -85,B 0,C 180,E1 -2987.234,E2 -2987.234} C_VEL
LIN {X 0,Y 560.734,Z 519.31,A -85,B 0,C 180,E1 -2988.258,E2 -2988.258} C_VEL
LIN {X 0,Y 561.131,Z 504.078,A -85,B 0,C 180,E1 -2989.192,E2 -2989.192} C_VEL
LIN {X 0,Y 561.491,Z 488.874,A -85,B 0,C 180,E1 -2989.954,E2 -2989.954} C_VEL
LIN {X 0,Y 561.816,Z 472.713,A -85,B 0,C 180,E1 -2990.596,E2 -2990.596} C_VEL
LIN {X 0,Y 562.102,Z 456.368,A -85,B 0,C 180,E1 -2991.088,E2 -2991.088} C_VEL
LIN {X 0,Y 562.282,Z 441.108,A -85,B 0,C 180,E1 -2991.418,E2 -2991.418} C_VEL
LIN {X 0,Y 563.186,Z 244.124,A -85,B 0,C 180,E1 -2994.066,E2 -2994.066} C_VEL
LIN {X 0,Y 561.61,Z 234.597,A -85,B 0,C 180,E1 -2994.291,E2 -2994.291} C_VEL
LIN {X 0,Y 562.27,Z 201.337,A -85,B 0,C 180,E1 -2997.229,E2 -2997.229} C_VEL
LIN {X 0,Y 561.942,Z 197.847,A -85,B 0,C 180,E1 -2997.561,E2 -2997.561} C_VEL
LIN {X 0,Y 559.161,Z 188.149,A -85,B 0,C 180,E1 -2998.603,E2 -2998.603} C_VEL
LIN {X 0,Y 559.132,Z 188.154,A -85,B 0,C 180,E1 -3001.271,E2 -3001.271} C_VEL
LIN {X 0,Y 559.149,Z 188.145,A -85,B 0,C 180,E1 -3003.947,E2 -3003.947} C_VEL
LIN {X 0,Y 559.121,Z 188.155,A -85,B 0,C 180,E1 -3007.106,E2 -3007.106} C_VEL
LIN {X 0,Y 559.143,Z 188.143,A -85,B 0,C 180,E1 -3009.94,E2 -3009.94} C_VEL
LIN {X 0,Y 559.137,Z 188.147,A -85,B 0,C 180,E1 -3012.741,E2 -3012.741} C_VEL
LIN {X 0,Y 559.129,Z 188.145,A -85,B 0,C 180,E1 -3015.759,E2 -3015.759} C_VEL
LIN {X 0,Y 559.167,Z 188.14,A -85,B 0,C 180,E1 -3018.231,E2 -3018.231} C_VEL
LIN {X 0,Y 559.152,Z 188.15,A -85,B 0,C 180,E1 -3021.189,E2 -3021.189} C_VEL
LIN {X 0,Y 559.142,Z 188.142,A -85,B 0,C 180,E1 -3023.79,E2 -3023.79} C_VEL
LIN {X 0,Y 559.133,Z 188.146,A -85,B 0,C 180,E1 -3026.423,E2 -3026.423} C_VEL
LIN {X 0,Y 559.134,Z 188.15,A -85,B 0,C 180,E1 -3028.98,E2 -3028.98} C_VEL
LIN {X 0,Y 559.162,Z 188.141,A -85,B 0,C 180,E1 -3032.287,E2 -3032.287} C_VEL
LIN {X 0,Y 559.146,Z 188.146,A -85,B 0,C 180,E1 -3034.812,E2 -3034.812} C_VEL
LIN {X 0,Y 559.143,Z 188.15,A -85,B 0,C 180,E1 -3037.068,E2 -3037.068} C_VEL
LIN {X 0,Y 559.156,Z 188.139,A -85,B 0,C 180,E1 -3039.395,E2 -3039.395} C_VEL
LIN {X 0,Y 559.132,Z 188.146,A -85,B 0,C 180,E1 -3042.443,E2 -3042.443} C_VEL
LIN {X 0,Y 559.16,Z 188.14,A -85,B 0,C 180,E1 -3045.441,E2 -3045.441} C_VEL
LIN {X 0,Y 559.202,Z 188.134,A -85,B 0,C 180,E1 -3048.588,E2 -3048.588} C_VEL
LIN {X 0,Y 559.16,Z 188.143,A -85,B 0,C 180,E1 -3051.326,E2 -3051.326} C_VEL
LIN {X 0,Y 559.201,Z 188.137,A -85,B 0,C 180,E1 -3054.23,E2 -3054.23} C_VEL
LIN {X 0,Y 559.212,Z 188.134,A -85,B 0,C 180,E1 -3057.119,E2 -3057.119} C_VEL
LIN {X 0,Y 559.219,Z 188.134,A -85,B 0,C 180,E1 -3060,E2 -3060} C_VEL
LIN {X 0,Y 559.217,Z 188.137,A -85,B 0,C 180,E1 -3062.882,E2 -3062.882} C_VEL
LIN {X 0,Y 559.194,Z 188.134,A -85,B 0,C 180,E1 -3065.771,E2 -3065.771} C_VEL
LIN {X 0,Y 559.171,Z 188.147,A -85,B 0,C 180,E1 -3068.675,E2 -3068.675} C_VEL
LIN {X 0,Y 559.175,Z 188.134,A -85,B 0,C 180,E1 -3071.601,E2 -3071.601} C_VEL
LIN {X 0,Y 559.166,Z 188.149,A -85,B 0,C 180,E1 -3074.597,E2 -3074.597} C_VEL
LIN {X 0,Y 559.164,Z 188.138,A -85,B 0,C 180,E1 -3077.557,E2 -3077.557} C_VEL
LIN {X 0,Y 559.16,Z 188.148,A -85,B 0,C 180,E1 -3080.606,E2 -3080.606} C_VEL
LIN {X 0,Y 559.136,Z 188.144,A -85,B 0,C 180,E1 -3083.718,E2 -3083.718} C_VEL
LIN {X 0,Y 559.151,Z 188.143,A -85,B 0,C 180,E1 -3086.099,E2 -3086.099} C_VEL
LIN {X 0,Y 559.139,Z 188.151,A -85,B 0,C 180,E1 -3088.531,E2 -3088.531} C_VEL
LIN {X 0,Y 559.112,Z 188.148,A -85,B 0,C 180,E1 -3090.651,E2 -3090.651} C_VEL
LIN {X 0,Y 558.452,Z 188.23,A -85,B 0,C 180,E1 -3091.253,E2 -3091.253} C_VEL
LIN {X 0,Y 555.588,Z 188.592,A -85,B 0,C 180,E1 -3092.229,E2 -3092.229} C_VEL
LIN {X 0,Y 553.175,Z 188.886,A -85,B 0,C 180,E1 -3093.015,E2 -3093.015} C_VEL
LIN {X 0,Y 552.158,Z 189.01,A -85,B 0,C 180,E1 -3093.622,E2 -3093.622} C_VEL
LIN {X 0,Y 552.085,Z 189.021,A -85,B 0,C 180,E1 -3093.827,E2 -3093.827} C_VEL
LIN {X 0,Y 552.086,Z 189.025,A -85,B 0,C 180,E1 -3096.749,E2 -3096.749} C_VEL
LIN {X 0,Y 552.105,Z 189.016,A -85,B 0,C 180,E1 -3099.53,E2 -3099.53} C_VEL
LIN {X 0,Y 552.11,Z 189.026,A -85,B 0,C 180,E1 -3102.428,E2 -3102.428} C_VEL
LIN {X 0,Y 552.073,Z 189.021,A -85,B 0,C 180,E1 -3105.565,E2 -3105.565} C_VEL
LIN {X 0,Y 552.102,Z 189.022,A -85,B 0,C 180,E1 -3108.681,E2 -3108.681} C_VEL
LIN {X 0,Y 552.099,Z 189.019,A -85,B 0,C 180,E1 -3111.414,E2 -3111.414} C_VEL
LIN {X 0,Y 552.087,Z 189.029,A -85,B 0,C 180,E1 -3114.16,E2 -3114.16} C_VEL
LIN {X 0,Y 552.103,Z 189.021,A -85,B 0,C 180,E1 -3116.817,E2 -3116.817} C_VEL
LIN {X 0,Y 552.089,Z 189.022,A -85,B 0,C 180,E1 -3119.393,E2 -3119.393} C_VEL
LIN {X 0,Y 552.069,Z 189.031,A -85,B 0,C 180,E1 -3121.903,E2 -3121.903} C_VEL
LIN {X 0,Y 552.077,Z 189.024,A -85,B 0,C 180,E1 -3124.668,E2 -3124.668} C_VEL
LIN {X 0,Y 552.079,Z 189.025,A -85,B 0,C 180,E1 -3127.551,E2 -3127.551} C_VEL
LIN {X 0,Y 552.135,Z 189.016,A -85,B 0,C 180,E1 -3130.676,E2 -3130.676} C_VEL
LIN {X 0,Y 552.072,Z 189.031,A -85,B 0,C 180,E1 -3133.738,E2 -3133.738} C_VEL
LIN {X 0,Y 552.121,Z 189.025,A -85,B 0,C 180,E1 -3136.006,E2 -3136.006} C_VEL
LIN {X 0,Y 552.16,Z 189.014,A -85,B 0,C 180,E1 -3138.996,E2 -3138.996} C_VEL
LIN {X 0,Y 552.113,Z 189.027,A -85,B 0,C 180,E1 -3141.953,E2 -3141.953} C_VEL
LIN {X 0,Y 552.209,Z 189.005,A -85,B 0,C 180,E1 -3144.891,E2 -3144.891} C_VEL
LIN {X 0,Y 552.222,Z 189.014,A -85,B 0,C 180,E1 -3147.814,E2 -3147.814} C_VEL
LIN {X 0,Y 552.096,Z 189.029,A -85,B 0,C 180,E1 -3150.503,E2 -3150.503} C_VEL
LIN {X 0,Y 554.596,Z 198.278,A -85,B 0,C 180,E1 -3151.636,E2 -3151.636} C_VEL
LIN {X 0,Y 554.79,Z 201.674,A -85,B 0,C 180,E1 -3151.998,E2 -3151.998} C_VEL
LIN {X 0,Y 554.736,Z 206.474,A -85,B 0,C 180,E1 -3152.475,E2 -3152.475} C_VEL
LIN {X 0,Y 556.64,Z 215.883,A -85,B 0,C 180,E1 -3152.697,E2 -3152.697} C_VEL
LIN {X 0,Y 555.856,Z 376.362,A -85,B 0,C 180,E1 -3154.875,E2 -3154.875} C_VEL
LIN {X 0,Y 555.654,Z 411.978,A -85,B 0,C 180,E1 -3155.377,E2 -3155.377} C_VEL
LIN {X 0,Y 555.43,Z 428.404,A -85,B 0,C 180,E1 -3155.743,E2 -3155.743} C_VEL
LIN {X 0,Y 555.133,Z 443.827,A -85,B 0,C 180,E1 -3156.225,E2 -3156.225} C_VEL
LIN {X 0,Y 554.791,Z 459.433,A -85,B 0,C 180,E1 -3156.868,E2 -3156.868} C_VEL
LIN {X 0,Y 554.348,Z 474.752,A -85,B 0,C 180,E1 -3157.651,E2 -3157.651} C_VEL
LIN {X 0,Y 553.924,Z 489.549,A -85,B 0,C 180,E1 -3158.573,E2 -3158.573} C_VEL
LIN {X 0,Y 553.514,Z 503.294,A -85,B 0,C 180,E1 -3159.594,E2 -3159.594} C_VEL
LIN {X 0,Y 553.164,Z 515.065,A -85,B 0,C 180,E1 -3160.617,E2 -3160.617} C_VEL
LIN {X 0,Y 552.777,Z 527.709,A -85,B 0,C 180,E1 -3161.906,E2 -3161.906} C_VEL
LIN {X 0,Y 552.432,Z 538.842,A -85,B 0,C 180,E1 -3163.239,E2 -3163.239} C_VEL
LIN {X 0,Y 552.193,Z 549.515,A -85,B 0,C 180,E1 -3164.748,E2 -3164.748} C_VEL
LIN {X 0,Y 552.005,Z 558.541,A -85,B 0,C 180,E1 -3166.267,E2 -3166.267} C_VEL
LIN {X 0,Y 551.888,Z 566.121,A -85,B 0,C 180,E1 -3167.797,E2 -3167.797} C_VEL
LIN {X 0,Y 551.833,Z 572.372,A -85,B 0,C 180,E1 -3169.338,E2 -3169.338} C_VEL
LIN {X 0,Y 551.756,Z 577.381,A -85,B 0,C 180,E1 -3170.896,E2 -3170.896} C_VEL
LIN {X 0,Y 551.658,Z 581.263,A -85,B 0,C 180,E1 -3172.471,E2 -3172.471} C_VEL
LIN {X 0,Y 551.602,Z 583.994,A -85,B 0,C 180,E1 -3174.062,E2 -3174.062} C_VEL
LIN {X 0,Y 551.625,Z 585.533,A -85,B 0,C 180,E1 -3175.67,E2 -3175.67} C_VEL
LIN {X 0,Y 551.632,Z 585.951,A -85,B 0,C 180,E1 -3177.301,E2 -3177.301} C_VEL
LIN {X 0,Y 551.651,Z 585.184,A -85,B 0,C 180,E1 -3178.955,E2 -3178.955} C_VEL
LIN {X 0,Y 551.685,Z 583.076,A -85,B 0,C 180,E1 -3180.636,E2 -3180.636} C_VEL
LIN {X 0,Y 551.693,Z 579.61,A -85,B 0,C 180,E1 -3182.347,E2 -3182.347} C_VEL
LIN {X 0,Y 551.748,Z 574.57,A -85,B 0,C 180,E1 -3184.11,E2 -3184.11} C_VEL
LIN {X 0,Y 551.865,Z 567.986,A -85,B 0,C 180,E1 -3185.861,E2 -3185.861} C_VEL
LIN {X 0,Y 551.975,Z 560.563,A -85,B 0,C 180,E1 -3187.444,E2 -3187.444} C_VEL
LIN {X 0,Y 552.15,Z 552.774,A -85,B 0,C 180,E1 -3188.827,E2 -3188.827} C_VEL
LIN {X 0,Y 552.33,Z 543.463,A -85,B 0,C 180,E1 -3190.229,E2 -3190.229} C_VEL
LIN {X 0,Y 552.597,Z 532.411,A -85,B 0,C 180,E1 -3191.646,E2 -3191.646} C_VEL
LIN {X 0,Y 552.977,Z 521.178,A -85,B 0,C 180,E1 -3192.875,E2 -3192.875} C_VEL
LIN {X 0,Y 553.374,Z 508.007,A -85,B 0,C 180,E1 -3194.106,E2 -3194.106} C_VEL
LIN {X 0,Y 553.802,Z 494.12,A -85,B 0,C 180,E1 -3195.2,E2 -3195.2} C_VEL
LIN {X 0,Y 554.215,Z 480.134,A -85,B 0,C 180,E1 -3196.124,E2 -3196.124} C_VEL
LIN {X 0,Y 554.576,Z 465.955,A -85,B 0,C 180,E1 -3196.909,E2 -3196.909} C_VEL
LIN {X 0,Y 554.991,Z 450.708,A -85,B 0,C 180,E1 -3197.599,E2 -3197.599} C_VEL
LIN {X 0,Y 555.296,Z 434.701,A -85,B 0,C 180,E1 -3198.17,E2 -3198.17} C_VEL
LIN {X 0,Y 555.638,Z 417.878,A -85,B 0,C 180,E1 -3198.6,E2 -3198.6} C_VEL
LIN {X 0,Y 555.775,Z 399.474,A -85,B 0,C 180,E1 -3198.903,E2 -3198.903} C_VEL
LIN {X 0,Y 556.721,Z 216.342,A -85,B 0,C 180,E1 -3201.384,E2 -3201.384} C_VEL
LIN {X 0,Y 554.726,Z 206.308,A -85,B 0,C 180,E1 -3201.625,E2 -3201.625} C_VEL
LIN {X 0,Y 554.808,Z 199.221,A -85,B 0,C 180,E1 -3202.357,E2 -3202.357} C_VEL
LIN {X 0,Y 552.128,Z 189.024,A -85,B 0,C 180,E1 -3203.583,E2 -3203.583} C_VEL
LIN {X 0,Y 552.131,Z 189.024,A -85,B 0,C 180,E1 -3205.939,E2 -3205.939} C_VEL
LIN {X 0,Y 552.121,Z 189.025,A -85,B 0,C 180,E1 -3208.54,E2 -3208.54} C_VEL
LIN {X 0,Y 552.126,Z 189.019,A -85,B 0,C 180,E1 -3211.437,E2 -3211.437} C_VEL
LIN {X 0,Y 552.13,Z 189.025,A -85,B 0,C 180,E1 -3214.355,E2 -3214.355} C_VEL
LIN {X 0,Y 552.099,Z 189.023,A -85,B 0,C 180,E1 -3216.757,E2 -3216.757} C_VEL
LIN {X 0,Y 552.119,Z 189.017,A -85,B 0,C 180,E1 -3219.119,E2 -3219.119} C_VEL
LIN {X 0,Y 552.127,Z 189.02,A -85,B 0,C 180,E1 -3221.444,E2 -3221.444} C_VEL
LIN {X 0,Y 552.115,Z 189.023,A -85,B 0,C 180,E1 -3223.737,E2 -3223.737} C_VEL
LIN {X 0,Y 552.133,Z 189.025,A -85,B 0,C 180,E1 -3226.004,E2 -3226.004} C_VEL
LIN {X 0,Y 552.16,Z 189.013,A -85,B 0,C 180,E1 -3228.993,E2 -3228.993} C_VEL
LIN {X 0,Y 552.154,Z 189.022,A -85,B 0,C 180,E1 -3231.951,E2 -3231.951} C_VEL
LIN {X 0,Y 552.223,Z 189.005,A -85,B 0,C 180,E1 -3234.889,E2 -3234.889} C_VEL
LIN {X 0,Y 552.216,Z 189.014,A -85,B 0,C 180,E1 -3237.811,E2 -3237.811} C_VEL
LIN {X 0,Y 552.237,Z 189.004,A -85,B 0,C 180,E1 -3240.729,E2 -3240.729} C_VEL
LIN {X 0,Y 552.2,Z 189.009,A -85,B 0,C 180,E1 -3242.918,E2 -3242.918} C_VEL
LIN {X 0,Y 552.192,Z 189.015,A -85,B 0,C 180,E1 -3245.844,E2 -3245.844} C_VEL
LIN {X 0,Y 552.14,Z 189.016,A -85,B 0,C 180,E1 -3248.786,E2 -3248.786} C_VEL
LIN {X 0,Y 552.159,Z 189.019,A -85,B 0,C 180,E1 -3251.75,E2 -3251.75} C_VEL
LIN {X 0,Y 552.133,Z 189.017,A -85,B 0,C 180,E1 -3254.748,E2 -3254.748} C_VEL
LIN {X 0,Y 552.095,Z 189.025,A -85,B 0,C 180,E1 -3257.789,E2 -3257.789} C_VEL
LIN {X 0,Y 552.122,Z 189.019,A -85,B 0,C 180,E1 -3260.101,E2 -3260.101} C_VEL
LIN {X 0,Y 552.088,Z 189.022,A -85,B 0,C 180,E1 -3262.451,E2 -3262.451} C_VEL
LIN {X 0,Y 552.134,Z 189.025,A -85,B 0,C 180,E1 -3265.346,E2 -3265.346} C_VEL
LIN {X 0,Y 552.093,Z 189.022,A -85,B 0,C 180,E1 -3268.099,E2 -3268.099} C_VEL
LIN {X 0,Y 552.096,Z 189.023,A -85,B 0,C 180,E1 -3270.609,E2 -3270.609} C_VEL
LIN {X 0,Y 552.104,Z 189.029,A -85,B 0,C 180,E1 -3273.186,E2 -3273.186} C_VEL
LIN {X 0,Y 552.083,Z 189.023,A -85,B 0,C 180,E1 -3275.844,E2 -3275.844} C_VEL
LIN {X 0,Y 552.117,Z 189.027,A -85,B 0,C 180,E1 -3279.061,E2 -3279.061} C_VEL
LIN {X 0,Y 552.118,Z 189.021,A -85,B 0,C 180,E1 -3281.446,E2 -3281.446} C_VEL
LIN {X 0,Y 552.074,Z 189.027,A -85,B 0,C 180,E1 -3284.529,E2 -3284.529} C_VEL
LIN {X 0,Y 552.107,Z 189.021,A -85,B 0,C 180,E1 -3287.587,E2 -3287.587} C_VEL
LIN {X 0,Y 552.13,Z 189.021,A -85,B 0,C 180,E1 -3290.472,E2 -3290.472} C_VEL
LIN {X 0,Y 552.099,Z 189.025,A -85,B 0,C 180,E1 -3293.318,E2 -3293.318} C_VEL
LIN {X 0,Y 552.125,Z 189.019,A -85,B 0,C 180,E1 -3295.938,E2 -3295.938} C_VEL
LIN {X 0,Y 552.121,Z 189.026,A -85,B 0,C 180,E1 -3298.54,E2 -3298.54} C_VEL
LIN {X 0,Y 552.099,Z 189.059,A -85,B 0,C 180,E1 -3301.125,E2 -3301.125} C_VEL
LIN {X 0,Y 555.586,Z 201.3,A -85,B 0,C 180,E1 -3302.44,E2 -3302.44} C_VEL
LIN {X 0,Y 554.924,Z 232.087,A -85,B 0,C 180,E1 -3305.195,E2 -3305.195} C_VEL
LIN {X 0,Y 554.854,Z 234.614,A -85,B 0,C 180,E1 -3305.418,E2 -3305.418} C_VEL
LIN {X 0,Y 556.705,Z 244.907,A -85,B 0,C 180,E1 -3305.651,E2 -3305.651} C_VEL
LIN {X 0,Y 555.661,Z 440.752,A -85,B 0,C 180,E1 -3308.311,E2 -3308.311} C_VEL
LIN {X 0,Y 555.453,Z 457.093,A -85,B 0,C 180,E1 -3308.667,E2 -3308.667} C_VEL
LIN {X 0,Y 555.117,Z 473.909,A -85,B 0,C 180,E1 -3309.188,E2 -3309.188} C_VEL
LIN {X 0,Y 554.827,Z 488.369,A -85,B 0,C 180,E1 -3309.772,E2 -3309.772} C_VEL
LIN {X 0,Y 554.392,Z 504.02,A -85,B 0,C 180,E1 -3310.562,E2 -3310.562} C_VEL
LIN {X 0,Y 553.931,Z 519.252,A -85,B 0,C 180,E1 -3311.506,E2 -3311.506} C_VEL
LIN {X 0,Y 553.476,Z 533.342,A -85,B 0,C 180,E1 -3312.554,E2 -3312.554} C_VEL
LIN {X 0,Y 553.047,Z 547.053,A -85,B 0,C 180,E1 -3313.764,E2 -3313.764} C_VEL
LIN {X 0,Y 552.737,Z 558.291,A -85,B 0,C 180,E1 -3314.924,E2 -3314.924} C_VEL
LIN {X 0,Y 552.446,Z 568.895,A -85,B 0,C 180,E1 -3316.199,E2 -3316.199} C_VEL
LIN {X 0,Y 552.21,Z 579.43,A -85,B 0,C 180,E1 -3317.69,E2 -3317.69} C_VEL
LIN {X 0,Y 551.993,Z 588.268,A -85,B 0,C 180,E1 -3319.174,E2 -3319.174} C_VEL
LIN {X 0,Y 551.862,Z 594.849,A -85,B 0,C 180,E1 -3320.469,E2 -3320.469} C_VEL
LIN {X 0,Y 551.805,Z 602.46,A -85,B 0,C 180,E1 -3322.313,E2 -3322.313} C_VEL
LIN {X 0,Y 551.772,Z 608.244,A -85,B 0,C 180,E1 -3324.15,E2 -3324.15} C_VEL
LIN {X 0,Y 551.701,Z 611.632,A -85,B 0,C 180,E1 -3325.615,E2 -3325.615} C_VEL
LIN {X 0,Y 551.712,Z 614.088,A -85,B 0,C 180,E1 -3327.078,E2 -3327.078} C_VEL
LIN {X 0,Y 551.639,Z 615.478,A -85,B 0,C 180,E1 -3328.538,E2 -3328.538} C_VEL
LIN {X 0,Y 551.636,Z 616,A -85,B 0,C 180,E1 -3329.998,E2 -3329.998} C_VEL
LIN {X 0,Y 551.638,Z 615.48,A -85,B 0,C 180,E1 -3331.458,E2 -3331.458} C_VEL
LIN {X 0,Y 551.711,Z 614.091,A -85,B 0,C 180,E1 -3332.919,E2 -3332.919} C_VEL
LIN {X 0,Y 551.701,Z 611.638,A -85,B 0,C 180,E1 -3334.382,E2 -3334.382} C_VEL
LIN {X 0,Y 551.77,Z 608.256,A -85,B 0,C 180,E1 -3335.846,E2 -3335.846} C_VEL
LIN {X 0,Y 551.803,Z 602.475,A -85,B 0,C 180,E1 -3337.683,E2 -3337.683} C_VEL
LIN {X 0,Y 551.867,Z 594.866,A -85,B 0,C 180,E1 -3339.527,E2 -3339.527} C_VEL
LIN {X 0,Y 552.037,Z 587.279,A -85,B 0,C 180,E1 -3341.007,E2 -3341.007} C_VEL
LIN {X 0,Y 552.223,Z 578.224,A -85,B 0,C 180,E1 -3342.493,E2 -3342.493} C_VEL
LIN {X 0,Y 552.485,Z 567.44,A -85,B 0,C 180,E1 -3343.984,E2 -3343.984} C_VEL
LIN {X 0,Y 552.852,Z 556.458,A -85,B 0,C 180,E1 -3345.276,E2 -3345.276} C_VEL
LIN {X 0,Y 553.158,Z 544.164,A -85,B 0,C 180,E1 -3346.513,E2 -3346.513} C_VEL
LIN {X 0,Y 553.571,Z 530.666,A -85,B 0,C 180,E1 -3347.661,E2 -3347.661} C_VEL
LIN {X 0,Y 553.983,Z 516.453,A -85,B 0,C 180,E1 -3348.68,E2 -3348.68} C_VEL
LIN {X 0,Y 554.421,Z 502.317,A -85,B 0,C 180,E1 -3349.53,E2 -3349.53} C_VEL
LIN {X 0,Y 554.827,Z 487.348,A -85,B 0,C 180,E1 -3350.275,E2 -3350.275} C_VEL
LIN {X 0,Y 555.223,Z 471.412,A -85,B 0,C 180,E1 -3350.901,E2 -3350.901} C_VEL
LIN {X 0,Y 555.473,Z 455.407,A -85,B 0,C 180,E1 -3351.377,E2 -3351.377} C_VEL
LIN {X 0,Y 555.694,Z 439.493,A -85,B 0,C 180,E1 -3351.709,E2 -3351.709} C_VEL
LIN {X 0,Y 556.655,Z 244.408,A -85,B 0,C 180,E1 -3354.359,E2 -3354.359} C_VEL
LIN {X 0,Y 554.891,Z 234.562,A -85,B 0,C 180,E1 -3354.592,E2 -3354.592} C_VEL
LIN {X 0,Y 555.62,Z 201.544,A -85,B 0,C 180,E1 -3357.547,E2 -3357.547} C_VEL
LIN {X 0,Y 552.099,Z 189.03,A -85,B 0,C 180,E1 -3358.899,E2 -3358.899} C_VEL
LIN {X 0,Y 552.095,Z 189.027,A -85,B 0,C 180,E1 -3361.473,E2 -3361.473} C_VEL
LIN {X 0,Y 552.117,Z 189.02,A -85,B 0,C 180,E1 -3364.168,E2 -3364.168} C_VEL
LIN {X 0,Y 552.086,Z 189.027,A -85,B 0,C 180,E1 -3366.745,E2 -3366.745} C_VEL
LIN {X 0,Y 552.111,Z 189.023,A -85,B 0,C 180,E1 -3369.525,E2 -3369.525} C_VEL
LIN {X 0,Y 552.107,Z 189.02,A -85,B 0,C 180,E1 -3372.423,E2 -3372.423} C_VEL
LIN {X 0,Y 552.073,Z 189.026,A -85,B 0,C 180,E1 -3375.561,E2 -3375.561} C_VEL
LIN {X 0,Y 552.115,Z 189.022,A -85,B 0,C 180,E1 -3378.674,E2 -3378.674} C_VEL
LIN {X 0,Y 552.094,Z 189.026,A -85,B 0,C 180,E1 -3381.409,E2 -3381.409} C_VEL
LIN {X 0,Y 552.084,Z 189.021,A -85,B 0,C 180,E1 -3384.157,E2 -3384.157} C_VEL
LIN {X 0,Y 552.092,Z 189.028,A -85,B 0,C 180,E1 -3386.813,E2 -3386.813} C_VEL
LIN {X 0,Y 552.078,Z 189.027,A -85,B 0,C 180,E1 -3389.39,E2 -3389.39} C_VEL
LIN {X 0,Y 552.096,Z 189.021,A -85,B 0,C 180,E1 -3391.901,E2 -3391.901} C_VEL
LIN {X 0,Y 552.123,Z 189.018,A -85,B 0,C 180,E1 -3394.648,E2 -3394.648} C_VEL
LIN {X 0,Y 552.091,Z 189.023,A -85,B 0,C 180,E1 -3397.549,E2 -3397.549} C_VEL
LIN {X 0,Y 552.125,Z 189.018,A -85,B 0,C 180,E1 -3400.674,E2 -3400.674} C_VEL
LIN {X 0,Y 552.088,Z 189.022,A -85,B 0,C 180,E1 -3403.737,E2 -3403.737} C_VEL
LIN {X 0,Y 552.105,Z 189.018,A -85,B 0,C 180,E1 -3406.004,E2 -3406.004} C_VEL
LIN {X 0,Y 552.177,Z 189.015,A -85,B 0,C 180,E1 -3408.994,E2 -3408.994} C_VEL
LIN {X 0,Y 552.128,Z 189.017,A -85,B 0,C 180,E1 -3411.951,E2 -3411.951} C_VEL
LIN {X 0,Y 552.202,Z 189.008,A -85,B 0,C 180,E1 -3414.889,E2 -3414.889} C_VEL
LIN {X 0,Y 552.184,Z 189.005,A -85,B 0,C 180,E1 -3417.812,E2 -3417.812} C_VEL
LIN {X 0,Y 552.22,Z 189.014,A -85,B 0,C 180,E1 -3420.73,E2 -3420.73} C_VEL
LIN {X 0,Y 552.182,Z 189.012,A -85,B 0,C 180,E1 -3422.919,E2 -3422.919} C_VEL
LIN {X 0,Y 552.164,Z 189.01,A -85,B 0,C 180,E1 -3425.845,E2 -3425.845} C_VEL
LIN {X 0,Y 552.139,Z 189.021,A -85,B 0,C 180,E1 -3428.786,E2 -3428.786} C_VEL
LIN {X 0,Y 552.131,Z 189.011,A -85,B 0,C 180,E1 -3431.752,E2 -3431.752} C_VEL
LIN {X 0,Y 552.104,Z 189.026,A -85,B 0,C 180,E1 -3434.75,E2 -3434.75} C_VEL
LIN {X 0,Y 552.134,Z 189.014,A -85,B 0,C 180,E1 -3437.333,E2 -3437.333} C_VEL
LIN {X 0,Y 552.106,Z 189.019,A -85,B 0,C 180,E1 -3440.103,E2 -3440.103} C_VEL
LIN {X 0,Y 552.084,Z 189.032,A -85,B 0,C 180,E1 -3442.452,E2 -3442.452} C_VEL
LIN {X 0,Y 552.125,Z 189.013,A -85,B 0,C 180,E1 -3445.352,E2 -3445.352} C_VEL
LIN {X 0,Y 552.099,Z 189.023,A -85,B 0,C 180,E1 -3448.099,E2 -3448.099} C_VEL
LIN {X 0,Y 552.073,Z 189.027,A -85,B 0,C 180,E1 -3450.648,E2 -3450.648} C_VEL
LIN {X 0,Y 552.087,Z 189.018,A -85,B 0,C 180,E1 -3453.188,E2 -3453.188} C_VEL
LIN {X 0,Y 552.085,Z 189.021,A -85,B 0,C 180,E1 -3453.827,E2 -3453.827} C_VEL
LIN {X 0,Y 551.455,Z 189.109,A -85,B 0,C 180,E1 -3454.436,E2 -3454.436} C_VEL
LIN {X 0,Y 548.632,Z 189.459,A -85,B 0,C 180,E1 -3455.424,E2 -3455.424} C_VEL
LIN {X 0,Y 546.208,Z 189.762,A -85,B 0,C 180,E1 -3456.219,E2 -3456.219} C_VEL
LIN {X 0,Y 545.138,Z 189.889,A -85,B 0,C 180,E1 -3456.833,E2 -3456.833} C_VEL
LIN {X 0,Y 545.036,Z 189.9,A -85,B 0,C 180,E1 -3457.041,E2 -3457.041} C_VEL
LIN {X 0,Y 545.046,Z 189.902,A -85,B 0,C 180,E1 -3460.145,E2 -3460.145} C_VEL
LIN {X 0,Y 545.043,Z 189.902,A -85,B 0,C 180,E1 -3462.699,E2 -3462.699} C_VEL
LIN {X 0,Y 545.03,Z 189.901,A -85,B 0,C 180,E1 -3465.873,E2 -3465.873} C_VEL
LIN {X 0,Y 545.063,Z 189.897,A -85,B 0,C 180,E1 -3468.888,E2 -3468.888} C_VEL
LIN {X 0,Y 545.062,Z 189.896,A -85,B 0,C 180,E1 -3470.821,E2 -3470.821} C_VEL
LIN {X 0,Y 545.035,Z 189.903,A -85,B 0,C 180,E1 -3473.623,E2 -3473.623} C_VEL
LIN {X 0,Y 545.053,Z 189.904,A -85,B 0,C 180,E1 -3476.331,E2 -3476.331} C_VEL
LIN {X 0,Y 545.055,Z 189.897,A -85,B 0,C 180,E1 -3478.955,E2 -3478.955} C_VEL
LIN {X 0,Y 545.066,Z 189.898,A -85,B 0,C 180,E1 -3481.509,E2 -3481.509} C_VEL
LIN {X 0,Y 545.03,Z 189.903,A -85,B 0,C 180,E1 -3484.507,E2 -3484.507} C_VEL
LIN {X 0,Y 545.024,Z 189.902,A -85,B 0,C 180,E1 -3487.245,E2 -3487.245} C_VEL
LIN {X 0,Y 545.099,Z 189.895,A -85,B 0,C 180,E1 -3490.417,E2 -3490.417} C_VEL
LIN {X 0,Y 545.02,Z 189.906,A -85,B 0,C 180,E1 -3493.522,E2 -3493.522} C_VEL
LIN {X 0,Y 545.078,Z 189.903,A -85,B 0,C 180,E1 -3495.822,E2 -3495.822} C_VEL
LIN {X 0,Y 545.117,Z 189.891,A -85,B 0,C 180,E1 -3498.852,E2 -3498.852} C_VEL
LIN {X 0,Y 545.07,Z 189.904,A -85,B 0,C 180,E1 -3501.848,E2 -3501.848} C_VEL
LIN {X 0,Y 545.167,Z 189.882,A -85,B 0,C 180,E1 -3504.825,E2 -3504.825} C_VEL
LIN {X 0,Y 545.194,Z 189.889,A -85,B 0,C 180,E1 -3507.786,E2 -3507.786} C_VEL
LIN {X 0,Y 545.165,Z 190.027,A -85,B 0,C 180,E1 -3510.256,E2 -3510.256} C_VEL
LIN {X 0,Y 548.135,Z 201.69,A -85,B 0,C 180,E1 -3511.655,E2 -3511.655} C_VEL
LIN {X 0,Y 548.123,Z 206.801,A -85,B 0,C 180,E1 -3512.16,E2 -3512.16} C_VEL
LIN {X 0,Y 550.17,Z 216.86,A -85,B 0,C 180,E1 -3512.403,E2 -3512.403} C_VEL
LIN {X 0,Y 549.523,Z 332.439,A -85,B 0,C 180,E1 -3513.994,E2 -3513.994} C_VEL
LIN {X 0,Y 549.098,Z 411.568,A -85,B 0,C 180,E1 -3515.096,E2 -3515.096} C_VEL
LIN {X 0,Y 548.828,Z 428.256,A -85,B 0,C 180,E1 -3515.467,E2 -3515.467} C_VEL
LIN {X 0,Y 548.471,Z 444.38,A -85,B 0,C 180,E1 -3515.978,E2 -3515.978} C_VEL
LIN {X 0,Y 548.087,Z 459.967,A -85,B 0,C 180,E1 -3516.629,E2 -3516.629} C_VEL
LIN {X 0,Y 547.646,Z 474.339,A -85,B 0,C 180,E1 -3517.375,E2 -3517.375} C_VEL
LIN {X 0,Y 547.147,Z 488.781,A -85,B 0,C 180,E1 -3518.278,E2 -3518.278} C_VEL
LIN {X 0,Y 546.756,Z 501.832,A -85,B 0,C 180,E1 -3519.247,E2 -3519.247} C_VEL
LIN {X 0,Y 546.269,Z 514.78,A -85,B 0,C 180,E1 -3520.378,E2 -3520.378} C_VEL
LIN {X 0,Y 545.866,Z 526.525,A -85,B 0,C 180,E1 -3521.58,E2 -3521.58} C_VEL
LIN {X 0,Y 545.532,Z 537.16,A -85,B 0,C 180,E1 -3522.841,E2 -3522.841} C_VEL
LIN {X 0,Y 545.272,Z 546.862,A -85,B 0,C 180,E1 -3524.177,E2 -3524.177} C_VEL
LIN {X 0,Y 545.013,Z 556.297,A -85,B 0,C 180,E1 -3525.713,E2 -3525.713} C_VEL
LIN {X 0,Y 544.832,Z 564.582,A -85,B 0,C 180,E1 -3527.338,E2 -3527.338} C_VEL
LIN {X 0,Y 544.737,Z 570.798,A -85,B 0,C 180,E1 -3528.818,E2 -3528.818} C_VEL
LIN {X 0,Y 544.683,Z 576.174,A -85,B 0,C 180,E1 -3530.389,E2 -3530.389} C_VEL
LIN {X 0,Y 544.555,Z 580.338,A -85,B 0,C 180,E1 -3531.98,E2 -3531.98} C_VEL
LIN {X 0,Y 544.519,Z 583.357,A -85,B 0,C 180,E1 -3533.596,E2 -3533.596} C_VEL
LIN {X 0,Y 544.527,Z 585.361,A -85,B 0,C 180,E1 -3535.382,E2 -3535.382} C_VEL
LIN {X 0,Y 544.543,Z 586,A -85,B 0,C 180,E1 -3537.059,E2 -3537.059} C_VEL
LIN {X 0,Y 544.561,Z 585.401,A -85,B 0,C 180,E1 -3538.645,E2 -3538.645} C_VEL
LIN {X 0,Y 544.601,Z 583.768,A -85,B 0,C 180,E1 -3540.219,E2 -3540.219} C_VEL
LIN {X 0,Y 544.576,Z 580.722,A -85,B 0,C 180,E1 -3541.947,E2 -3541.947} C_VEL
LIN {X 0,Y 544.677,Z 576.174,A -85,B 0,C 180,E1 -3543.7,E2 -3543.7} C_VEL
LIN {X 0,Y 544.791,Z 569.982,A -85,B 0,C 180,E1 -3545.487,E2 -3545.487} C_VEL
LIN {X 0,Y 544.879,Z 563.883,A -85,B 0,C 180,E1 -3546.898,E2 -3546.898} C_VEL
LIN {X 0,Y 545.047,Z 555.731,A -85,B 0,C 180,E1 -3548.474,E2 -3548.474} C_VEL
LIN {X 0,Y 545.247,Z 546.887,A -85,B 0,C 180,E1 -3549.91,E2 -3549.91} C_VEL
LIN {X 0,Y 545.549,Z 536.829,A -85,B 0,C 180,E1 -3551.292,E2 -3551.292} C_VEL
LIN {X 0,Y 545.886,Z 526.385,A -85,B 0,C 180,E1 -3552.525,E2 -3552.525} C_VEL
LIN {X 0,Y 546.28,Z 514.812,A -85,B 0,C 180,E1 -3553.709,E2 -3553.709} C_VEL
LIN {X 0,Y 546.741,Z 501.624,A -85,B 0,C 180,E1 -3554.861,E2 -3554.861} C_VEL
LIN {X 0,Y 547.19,Z 488.085,A -85,B 0,C 180,E1 -3555.861,E2 -3555.861} C_VEL
LIN {X 0,Y 547.634,Z 473.826,A -85,B 0,C 180,E1 -3556.747,E2 -3556.747} C_VEL
LIN {X 0,Y 548.103,Z 458.296,A -85,B 0,C 180,E1 -3557.539,E2 -3557.539} C_VEL
LIN {X 0,Y 548.521,Z 443.256,A -85,B 0,C 180,E1 -3558.153,E2 -3558.153} C_VEL
LIN {X 0,Y 548.846,Z 427.214,A -85,B 0,C 180,E1 -3558.652,E2 -3558.652} C_VEL
LIN {X 0,Y 549.116,Z 410.232,A -85,B 0,C 180,E1 -3559.019,E2 -3559.019} C_VEL
LIN {X 0,Y 550.255,Z 217.083,A -85,B 0,C 180,E1 -3561.681,E2 -3561.681} C_VEL
LIN {X 0,Y 548.054,Z 206.417,A -85,B 0,C 180,E1 -3561.958,E2 -3561.958} C_VEL
LIN {X 0,Y 548.157,Z 201.363,A -85,B 0,C 180,E1 -3562.482,E2 -3562.482} C_VEL
LIN {X 0,Y 545.067,Z 189.906,A -85,B 0,C 180,E1 -3563.885,E2 -3563.885} C_VEL
LIN {X 0,Y 545.069,Z 189.904,A -85,B 0,C 180,E1 -3566.328,E2 -3566.328} C_VEL
LIN {X 0,Y 545.067,Z 189.9,A -85,B 0,C 180,E1 -3568.952,E2 -3568.952} C_VEL
LIN {X 0,Y 545.104,Z 189.894,A -85,B 0,C 180,E1 -3571.507,E2 -3571.507} C_VEL
LIN {X 0,Y 545.095,Z 189.9,A -85,B 0,C 180,E1 -3574.491,E2 -3574.491} C_VEL
LIN {X 0,Y 545.037,Z 189.902,A -85,B 0,C 180,E1 -3577.242,E2 -3577.242} C_VEL
LIN {X 0,Y 545.12,Z 189.895,A -85,B 0,C 180,E1 -3580.414,E2 -3580.414} C_VEL
LIN {X 0,Y 545.072,Z 189.897,A -85,B 0,C 180,E1 -3583.521,E2 -3583.521} C_VEL
LIN {X 0,Y 545.093,Z 189.901,A -85,B 0,C 180,E1 -3585.819,E2 -3585.819} C_VEL
LIN {X 0,Y 545.115,Z 189.891,A -85,B 0,C 180,E1 -3588.849,E2 -3588.849} C_VEL
LIN {X 0,Y 545.124,Z 189.897,A -85,B 0,C 180,E1 -3591.847,E2 -3591.847} C_VEL
LIN {X 0,Y 545.199,Z 189.88,A -85,B 0,C 180,E1 -3594.822,E2 -3594.822} C_VEL
LIN {X 0,Y 545.189,Z 189.89,A -85,B 0,C 180,E1 -3597.783,E2 -3597.783} C_VEL
LIN {X 0,Y 545.208,Z 189.879,A -85,B 0,C 180,E1 -3600.738,E2 -3600.738} C_VEL
LIN {X 0,Y 545.167,Z 189.885,A -85,B 0,C 180,E1 -3602.955,E2 -3602.955} C_VEL
LIN {X 0,Y 545.164,Z 189.889,A -85,B 0,C 180,E1 -3605.919,E2 -3605.919} C_VEL
LIN {X 0,Y 545.103,Z 189.894,A -85,B 0,C 180,E1 -3608.9,E2 -3608.9} C_VEL
LIN {X 0,Y 545.103,Z 189.896,A -85,B 0,C 180,E1 -3611.905,E2 -3611.905} C_VEL
LIN {X 0,Y 545.082,Z 189.897,A -85,B 0,C 180,E1 -3614.943,E2 -3614.943} C_VEL
LIN {X 0,Y 545.066,Z 189.898,A -85,B 0,C 180,E1 -3618.026,E2 -3618.026} C_VEL
LIN {X 0,Y 545.088,Z 189.894,A -85,B 0,C 180,E1 -3620.372,E2 -3620.372} C_VEL
LIN {X 0,Y 545.076,Z 189.9,A -85,B 0,C 180,E1 -3623.559,E2 -3623.559} C_VEL
LIN {X 0,Y 545.075,Z 189.896,A -85,B 0,C 180,E1 -3626,E2 -3626} C_VEL
LIN {X 0,Y 545.071,Z 189.899,A -85,B 0,C 180,E1 -3628.745,E2 -3628.745} C_VEL
LIN {X 0,Y 545.055,Z 189.9,A -85,B 0,C 180,E1 -3631.679,E2 -3631.679} C_VEL
LIN {X 0,Y 545.057,Z 189.899,A -85,B 0,C 180,E1 -3634.564,E2 -3634.564} C_VEL
LIN {X 0,Y 545.033,Z 189.907,A -85,B 0,C 180,E1 -3637.304,E2 -3637.304} C_VEL
LIN {X 0,Y 545.062,Z 189.898,A -85,B 0,C 180,E1 -3640.143,E2 -3640.143} C_VEL
LIN {X 0,Y 545.037,Z 189.905,A -85,B 0,C 180,E1 -3642.694,E2 -3642.694} C_VEL
LIN {X 0,Y 545.028,Z 189.91,A -85,B 0,C 180,E1 -3645.17,E2 -3645.17} C_VEL
LIN {X 0,Y 545.051,Z 189.898,A -85,B 0,C 180,E1 -3647.894,E2 -3647.894} C_VEL
LIN {X 0,Y 545.08,Z 189.902,A -85,B 0,C 180,E1 -3650.818,E2 -3650.818} C_VEL
LIN {X 0,Y 545.034,Z 189.903,A -85,B 0,C 180,E1 -3653.618,E2 -3653.618} C_VEL
LIN {X 0,Y 545.063,Z 189.902,A -85,B 0,C 180,E1 -3656.327,E2 -3656.327} C_VEL
LIN {X 0,Y 545.063,Z 189.904,A -85,B 0,C 180,E1 -3658.951,E2 -3658.951} C_VEL
LIN {X 0,Y 545.045,Z 189.927,A -85,B 0,C 180,E1 -3660.818,E2 -3660.818} C_VEL
LIN {X 0,Y 548.747,Z 202.521,A -85,B 0,C 180,E1 -3662.201,E2 -3662.201} C_VEL
LIN {X 0,Y 548.774,Z 210.685,A -85,B 0,C 180,E1 -3662.957,E2 -3662.957} C_VEL
LIN {X 0,Y 548.154,Z 234.28,A -85,B 0,C 180,E1 -3665.089,E2 -3665.089} C_VEL
LIN {X 0,Y 550.221,Z 246.334,A -85,B 0,C 180,E1 -3665.369,E2 -3665.369} C_VEL
LIN {X 0,Y 549.056,Z 438.796,A -85,B 0,C 180,E1 -3668.011,E2 -3668.011} C_VEL
LIN {X 0,Y 548.84,Z 455.812,A -85,B 0,C 180,E1 -3668.373,E2 -3668.373} C_VEL
LIN {X 0,Y 548.492,Z 472.311,A -85,B 0,C 180,E1 -3668.876,E2 -3668.876} C_VEL
LIN {X 0,Y 548.148,Z 486.557,A -85,B 0,C 180,E1 -3669.441,E2 -3669.441} C_VEL
LIN {X 0,Y 547.645,Z 502.139,A -85,B 0,C 180,E1 -3670.215,E2 -3670.215} C_VEL
LIN {X 0,Y 547.235,Z 516.379,A -85,B 0,C 180,E1 -3671.077,E2 -3671.077} C_VEL
LIN {X 0,Y 546.783,Z 529.675,A -85,B 0,C 180,E1 -3672.031,E2 -3672.031} C_VEL
LIN {X 0,Y 546.324,Z 543.098,A -85,B 0,C 180,E1 -3673.174,E2 -3673.174} C_VEL
LIN {X 0,Y 545.945,Z 554.491,A -85,B 0,C 180,E1 -3674.315,E2 -3674.315} C_VEL
LIN {X 0,Y 545.596,Z 565.925,A -85,B 0,C 180,E1 -3675.642,E2 -3675.642} C_VEL
LIN {X 0,Y 545.267,Z 575.729,A -85,B 0,C 180,E1 -3676.963,E2 -3676.963} C_VEL
LIN {X 0,Y 545.086,Z 585.276,A -85,B 0,C 180,E1 -3678.491,E2 -3678.491} C_VEL
LIN {X 0,Y 544.873,Z 593.042,A -85,B 0,C 180,E1 -3679.971,E2 -3679.971} C_VEL
LIN {X 0,Y 544.749,Z 599.619,A -85,B 0,C 180,E1 -3681.466,E2 -3681.466} C_VEL
LIN {X 0,Y 544.724,Z 604.952,A -85,B 0,C 180,E1 -3682.958,E2 -3682.958} C_VEL
LIN {X 0,Y 544.687,Z 608.245,A -85,B 0,C 180,E1 -3684.074,E2 -3684.074} C_VEL
LIN {X 0,Y 544.6,Z 611.631,A -85,B 0,C 180,E1 -3685.558,E2 -3685.558} C_VEL
LIN {X 0,Y 544.638,Z 614.088,A -85,B 0,C 180,E1 -3687.04,E2 -3687.04} C_VEL
LIN {X 0,Y 544.54,Z 615.478,A -85,B 0,C 180,E1 -3688.519,E2 -3688.519} C_VEL
LIN {X 0,Y 544.536,Z 616,A -85,B 0,C 180,E1 -3689.998,E2 -3689.998} C_VEL
LIN {X 0,Y 544.539,Z 615.479,A -85,B 0,C 180,E1 -3691.477,E2 -3691.477} C_VEL
LIN {X 0,Y 544.638,Z 614.092,A -85,B 0,C 180,E1 -3692.957,E2 -3692.957} C_VEL
LIN {X 0,Y 544.599,Z 611.638,A -85,B 0,C 180,E1 -3694.439,E2 -3694.439} C_VEL
LIN {X 0,Y 544.685,Z 608.257,A -85,B 0,C 180,E1 -3695.923,E2 -3695.923} C_VEL
LIN {X 0,Y 544.738,Z 602.475,A -85,B 0,C 180,E1 -3697.784,E2 -3697.784} C_VEL
LIN {X 0,Y 544.799,Z 594.866,A -85,B 0,C 180,E1 -3699.652,E2 -3699.652} C_VEL
LIN {X 0,Y 545.013,Z 587.279,A -85,B 0,C 180,E1 -3701.151,E2 -3701.151} C_VEL
LIN {X 0,Y 545.225,Z 578.223,A -85,B 0,C 180,E1 -3702.656,E2 -3702.656} C_VEL
LIN {X 0,Y 545.529,Z 567.439,A -85,B 0,C 180,E1 -3704.166,E2 -3704.166} C_VEL
LIN {X 0,Y 545.92,Z 556.307,A -85,B 0,C 180,E1 -3705.491,E2 -3705.491} C_VEL
LIN {X 0,Y 546.26,Z 544.162,A -85,B 0,C 180,E1 -3706.728,E2 -3706.728} C_VEL
LIN {X 0,Y 546.712,Z 531.384,A -85,B 0,C 180,E1 -3707.83,E2 -3707.83} C_VEL
LIN {X 0,Y 547.147,Z 517.867,A -85,B 0,C 180,E1 -3708.825,E2 -3708.825} C_VEL
LIN {X 0,Y 547.621,Z 503.988,A -85,B 0,C 180,E1 -3709.684,E2 -3709.684} C_VEL
LIN {X 0,Y 548.096,Z 487.981,A -85,B 0,C 180,E1 -3710.498,E2 -3710.498} C_VEL
LIN {X 0,Y 548.52,Z 472.451,A -85,B 0,C 180,E1 -3711.119,E2 -3711.119} C_VEL
LIN {X 0,Y 548.831,Z 456.008,A -85,B 0,C 180,E1 -3711.624,E2 -3711.624} C_VEL
LIN {X 0,Y 549.1,Z 439.103,A -85,B 0,C 180,E1 -3711.983,E2 -3711.983} C_VEL
LIN {X 0,Y 550.195,Z 245.475,A -85,B 0,C 180,E1 -3714.646,E2 -3714.646} C_VEL
LIN {X 0,Y 548.186,Z 234.436,A -85,B 0,C 180,E1 -3714.907,E2 -3714.907} C_VEL
LIN {X 0,Y 548.985,Z 204.33,A -85,B 0,C 180,E1 -3717.633,E2 -3717.633} C_VEL
LIN {X 0,Y 547.607,Z 198.573,A -85,B 0,C 180,E1 -3718.242,E2 -3718.242} C_VEL
LIN {X 0,Y 545.067,Z 189.906,A -85,B 0,C 180,E1 -3719.219,E2 -3719.219} C_VEL
LIN {X 0,Y 545.043,Z 189.9,A -85,B 0,C 180,E1 -3721.912,E2 -3721.912} C_VEL
LIN {X 0,Y 545.057,Z 189.901,A -85,B 0,C 180,E1 -3724.561,E2 -3724.561} C_VEL
LIN {X 0,Y 545.017,Z 189.91,A -85,B 0,C 180,E1 -3727.302,E2 -3727.302} C_VEL
LIN {X 0,Y 545.05,Z 189.898,A -85,B 0,C 180,E1 -3730.14,E2 -3730.14} C_VEL
LIN {X 0,Y 545.057,Z 189.904,A -85,B 0,C 180,E1 -3733.104,E2 -3733.104} C_VEL
LIN {X 0,Y 545.042,Z 189.899,A -85,B 0,C 180,E1 -3736.222,E2 -3736.222} C_VEL
LIN {X 0,Y 545.076,Z 189.902,A -85,B 0,C 180,E1 -3738.885,E2 -3738.885} C_VEL
LIN {X 0,Y 545.027,Z 189.903,A -85,B 0,C 180,E1 -3741.761,E2 -3741.761} C_VEL
LIN {X 0,Y 545.035,Z 189.901,A -85,B 0,C 180,E1 -3744.532,E2 -3744.532} C_VEL
LIN {X 0,Y 545.051,Z 189.901,A -85,B 0,C 180,E1 -3747.211,E2 -3747.211} C_VEL
LIN {X 0,Y 545.036,Z 189.901,A -85,B 0,C 180,E1 -3749.809,E2 -3749.809} C_VEL
LIN {X 0,Y 545.063,Z 189.898,A -85,B 0,C 180,E1 -3752.343,E2 -3752.343} C_VEL
LIN {X 0,Y 545.085,Z 189.897,A -85,B 0,C 180,E1 -3754.819,E2 -3754.819} C_VEL
LIN {X 0,Y 545.043,Z 189.904,A -85,B 0,C 180,E1 -3757.243,E2 -3757.243} C_VEL
LIN {X 0,Y 545.088,Z 189.891,A -85,B 0,C 180,E1 -3760.414,E2 -3760.414} C_VEL
LIN {X 0,Y 545.044,Z 189.901,A -85,B 0,C 180,E1 -3763.521,E2 -3763.521} C_VEL
LIN {X 0,Y 545.063,Z 189.895,A -85,B 0,C 180,E1 -3765.819,E2 -3765.819} C_VEL
LIN {X 0,Y 545.124,Z 189.891,A -85,B 0,C 180,E1 -3768.85,E2 -3768.85} C_VEL
LIN {X 0,Y 545.098,Z 189.893,A -85,B 0,C 180,E1 -3771.847,E2 -3771.847} C_VEL
LIN {X 0,Y 545.177,Z 189.883,A -85,B 0,C 180,E1 -3774.823,E2 -3774.823} C_VEL
LIN {X 0,Y 545.156,Z 189.88,A -85,B 0,C 180,E1 -3777.784,E2 -3777.784} C_VEL
LIN {X 0,Y 545.189,Z 189.89,A -85,B 0,C 180,E1 -3780.739,E2 -3780.739} C_VEL
LIN {X 0,Y 545.147,Z 189.888,A -85,B 0,C 180,E1 -3782.956,E2 -3782.956} C_VEL
LIN {X 0,Y 545.136,Z 189.885,A -85,B 0,C 180,E1 -3785.92,E2 -3785.92} C_VEL
LIN {X 0,Y 545.096,Z 189.896,A -85,B 0,C 180,E1 -3788.901,E2 -3788.901} C_VEL
LIN {X 0,Y 545.103,Z 189.887,A -85,B 0,C 180,E1 -3791.905,E2 -3791.905} C_VEL
LIN {X 0,Y 545.053,Z 189.901,A -85,B 0,C 180,E1 -3794.945,E2 -3794.945} C_VEL
LIN {X 0,Y 545.086,Z 189.891,A -85,B 0,C 180,E1 -3797.438,E2 -3797.438} C_VEL
LIN {X 0,Y 545.07,Z 189.899,A -85,B 0,C 180,E1 -3800.373,E2 -3800.373} C_VEL
LIN {X 0,Y 545.084,Z 189.894,A -85,B 0,C 180,E1 -3803.56,E2 -3803.56} C_VEL
LIN {X 0,Y 545.05,Z 189.897,A -85,B 0,C 180,E1 -3806.003,E2 -3806.003} C_VEL
LIN {X 0,Y 545.064,Z 189.901,A -85,B 0,C 180,E1 -3808.751,E2 -3808.751} C_VEL
LIN {X 0,Y 545.031,Z 189.9,A -85,B 0,C 180,E1 -3811.681,E2 -3811.681} C_VEL
LIN {X 0,Y 545.051,Z 189.904,A -85,B 0,C 180,E1 -3814.566,E2 -3814.566} C_VEL
LIN {X 0,Y 545.036,Z 189.9,A -85,B 0,C 180,E1 -3817.041,E2 -3817.041} C_VEL
LIN {X 0,Y 544.328,Z 189.99,A -85,B 0,C 180,E1 -3817.657,E2 -3817.657} C_VEL
LIN {X 0,Y 541.457,Z 190.345,A -85,B 0,C 180,E1 -3818.658,E2 -3818.658} C_VEL
LIN {X 0,Y 539.068,Z 190.64,A -85,B 0,C 180,E1 -3819.464,E2 -3819.464} C_VEL
LIN {X 0,Y 538.064,Z 190.77,A -85,B 0,C 180,E1 -3820.086,E2 -3820.086} C_VEL
LIN {X 0,Y 537.992,Z 190.775,A -85,B 0,C 180,E1 -3820.296,E2 -3820.296} C_VEL
LIN {X 0,Y 538.006,Z 190.776,A -85,B 0,C 180,E1 -3822.99,E2 -3822.99} C_VEL
LIN {X 0,Y 537.985,Z 190.783,A -85,B 0,C 180,E1 -3826.187,E2 -3826.187} C_VEL
LIN {X 0,Y 538.032,Z 190.772,A -85,B 0,C 180,E1 -3829.256,E2 -3829.256} C_VEL
LIN {X 0,Y 537.976,Z 190.787,A -85,B 0,C 180,E1 -3832.125,E2 -3832.125} C_VEL
LIN {X 0,Y 537.994,Z 190.775,A -85,B 0,C 180,E1 -3834.919,E2 -3834.919} C_VEL
LIN {X 0,Y 538.007,Z 190.779,A -85,B 0,C 180,E1 -3837.62,E2 -3837.62} C_VEL
LIN {X 0,Y 538.003,Z 190.782,A -85,B 0,C 180,E1 -3840.241,E2 -3840.241} C_VEL
LIN {X 0,Y 538.006,Z 190.777,A -85,B 0,C 180,E1 -3842.796,E2 -3842.796} C_VEL
LIN {X 0,Y 537.978,Z 190.78,A -85,B 0,C 180,E1 -3845.292,E2 -3845.292} C_VEL
LIN {X 0,Y 538.01,Z 190.783,A -85,B 0,C 180,E1 -3848.045,E2 -3848.045} C_VEL
LIN {X 0,Y 538.004,Z 190.776,A -85,B 0,C 180,E1 -3850.942,E2 -3850.942} C_VEL
LIN {X 0,Y 537.967,Z 190.783,A -85,B 0,C 180,E1 -3853.3,E2 -3853.3} C_VEL
LIN {X 0,Y 538.049,Z 190.777,A -85,B 0,C 180,E1 -3855.633,E2 -3855.633} C_VEL
LIN {X 0,Y 538.077,Z 190.769,A -85,B 0,C 180,E1 -3858.704,E2 -3858.704} C_VEL
LIN {X 0,Y 538.041,Z 190.78,A -85,B 0,C 180,E1 -3861.741,E2 -3861.741} C_VEL
LIN {X 0,Y 538.127,Z 190.759,A -85,B 0,C 180,E1 -3864.757,E2 -3864.757} C_VEL
LIN {X 0,Y 538.165,Z 190.765,A -85,B 0,C 180,E1 -3867.757,E2 -3867.757} C_VEL
LIN {X 0,Y 538.174,Z 190.92,A -85,B 0,C 180,E1 -3869.955,E2 -3869.955} C_VEL
LIN {X 0,Y 541.425,Z 203.488,A -85,B 0,C 180,E1 -3871.489,E2 -3871.489} C_VEL
LIN {X 0,Y 541.368,Z 206.535,A -85,B 0,C 180,E1 -3871.81,E2 -3871.81} C_VEL
LIN {X 0,Y 543.751,Z 218.131,A -85,B 0,C 180,E1 -3872.108,E2 -3872.108} C_VEL
LIN {X 0,Y 542.66,Z 392.117,A -85,B 0,C 180,E1 -3874.528,E2 -3874.528} C_VEL
LIN {X 0,Y 542.449,Z 415.08,A -85,B 0,C 180,E1 -3874.879,E2 -3874.879} C_VEL
LIN {X 0,Y 542.145,Z 432.181,A -85,B 0,C 180,E1 -3875.301,E2 -3875.301} C_VEL
LIN {X 0,Y 541.712,Z 448.56,A -85,B 0,C 180,E1 -3875.866,E2 -3875.866} C_VEL
LIN {X 0,Y 541.313,Z 463.385,A -85,B 0,C 180,E1 -3876.525,E2 -3876.525} C_VEL
LIN {X 0,Y 540.772,Z 478.841,A -85,B 0,C 180,E1 -3877.375,E2 -3877.375} C_VEL
LIN {X 0,Y 540.271,Z 492.896,A -85,B 0,C 180,E1 -3878.314,E2 -3878.314} C_VEL
LIN {X 0,Y 539.732,Z 506.172,A -85,B 0,C 180,E1 -3879.369,E2 -3879.369} C_VEL
LIN {X 0,Y 539.241,Z 518.472,A -85,B 0,C 180,E1 -3880.515,E2 -3880.515} C_VEL
LIN {X 0,Y 538.816,Z 530.216,A -85,B 0,C 180,E1 -3881.793,E2 -3881.793} C_VEL
LIN {X 0,Y 538.386,Z 541.343,A -85,B 0,C 180,E1 -3883.207,E2 -3883.207} C_VEL
LIN {X 0,Y 538.141,Z 550.756,A -85,B 0,C 180,E1 -3884.62,E2 -3884.62} C_VEL
LIN {X 0,Y 537.905,Z 559.258,A -85,B 0,C 180,E1 -3886.121,E2 -3886.121} C_VEL
LIN {X 0,Y 537.752,Z 565.882,A -85,B 0,C 180,E1 -3887.494,E2 -3887.494} C_VEL
LIN {X 0,Y 537.65,Z 572.152,A -85,B 0,C 180,E1 -3889.075,E2 -3889.075} C_VEL
LIN {X 0,Y 537.592,Z 577.205,A -85,B 0,C 180,E1 -3890.67,E2 -3890.67} C_VEL
LIN {X 0,Y 537.46,Z 581.143,A -85,B 0,C 180,E1 -3892.286,E2 -3892.286} C_VEL
LIN {X 0,Y 537.421,Z 583.896,A -85,B 0,C 180,E1 -3893.917,E2 -3893.917} C_VEL
LIN {X 0,Y 537.441,Z 585.49,A -85,B 0,C 180,E1 -3895.566,E2 -3895.566} C_VEL
LIN {X 0,Y 537.461,Z 585.966,A -85,B 0,C 180,E1 -3897.238,E2 -3897.238} C_VEL
LIN {X 0,Y 537.474,Z 585.232,A -85,B 0,C 180,E1 -3898.935,E2 -3898.935} C_VEL
LIN {X 0,Y 537.477,Z 583.177,A -85,B 0,C 180,E1 -3900.662,E2 -3900.662} C_VEL
LIN {X 0,Y 537.517,Z 579.772,A -85,B 0,C 180,E1 -3902.417,E2 -3902.417} C_VEL
LIN {X 0,Y 537.585,Z 574.865,A -85,B 0,C 180,E1 -3904.205,E2 -3904.205} C_VEL
LIN {X 0,Y 537.722,Z 568.917,A -85,B 0,C 180,E1 -3905.87,E2 -3905.87} C_VEL
LIN {X 0,Y 537.874,Z 561.748,A -85,B 0,C 180,E1 -3907.484,E2 -3907.484} C_VEL
LIN {X 0,Y 538.077,Z 553.468,A -85,B 0,C 180,E1 -3909.018,E2 -3909.018} C_VEL
LIN {X 0,Y 538.31,Z 543.961,A -85,B 0,C 180,E1 -3910.506,E2 -3910.506} C_VEL
LIN {X 0,Y 538.692,Z 533.029,A -85,B 0,C 180,E1 -3911.956,E2 -3911.956} C_VEL
LIN {X 0,Y 539.137,Z 522.377,A -85,B 0,C 180,E1 -3913.177,E2 -3913.177} C_VEL
LIN {X 0,Y 539.611,Z 509.96,A -85,B 0,C 180,E1 -3914.391,E2 -3914.391} C_VEL
LIN {X 0,Y 540.096,Z 496.939,A -85,B 0,C 180,E1 -3915.473,E2 -3915.473} C_VEL
LIN {X 0,Y 540.578,Z 483.165,A -85,B 0,C 180,E1 -3916.445,E2 -3916.445} C_VEL
LIN {X 0,Y 541.148,Z 468.215,A -85,B 0,C 180,E1 -3917.32,E2 -3917.32} C_VEL
LIN {X 0,Y 541.625,Z 452.979,A -85,B 0,C 180,E1 -3918.046,E2 -3918.046} C_VEL
LIN {X 0,Y 542.032,Z 436.393,A -85,B 0,C 180,E1 -3918.662,E2 -3918.662} C_VEL
LIN {X 0,Y 542.438,Z 419.23,A -85,B 0,C 180,E1 -3919.123,E2 -3919.123} C_VEL
LIN {X 0,Y 542.629,Z 402.099,A -85,B 0,C 180,E1 -3919.423,E2 -3919.423} C_VEL
LIN {X 0,Y 543.823,Z 218.304,A -85,B 0,C 180,E1 -3921.978,E2 -3921.978} C_VEL
LIN {X 0,Y 541.426,Z 206.808,A -85,B 0,C 180,E1 -3922.267,E2 -3922.267} C_VEL
LIN {X 0,Y 541.444,Z 203.298,A -85,B 0,C 180,E1 -3922.64,E2 -3922.64} C_VEL
LIN {X 0,Y 538.03,Z 190.783,A -85,B 0,C 180,E1 -3924.189,E2 -3924.189} C_VEL
LIN {X 0,Y 538.033,Z 190.779,A -85,B 0,C 180,E1 -3926.727,E2 -3926.727} C_VEL
LIN {X 0,Y 538.028,Z 190.777,A -85,B 0,C 180,E1 -3929.556,E2 -3929.556} C_VEL
LIN {X 0,Y 538.045,Z 190.777,A -85,B 0,C 180,E1 -3931.95,E2 -3931.95} C_VEL
LIN {X 0,Y 538.071,Z 190.775,A -85,B 0,C 180,E1 -3934.467,E2 -3934.467} C_VEL
LIN {X 0,Y 537.993,Z 190.784,A -85,B 0,C 180,E1 -3937.738,E2 -3937.738} C_VEL
LIN {X 0,Y 538.08,Z 190.776,A -85,B 0,C 180,E1 -3940.147,E2 -3940.147} C_VEL
LIN {X 0,Y 538.023,Z 190.773,A -85,B 0,C 180,E1 -3943.299,E2 -3943.299} C_VEL
LIN {X 0,Y 538.062,Z 190.774,A -85,B 0,C 180,E1 -3945.63,E2 -3945.63} C_VEL
LIN {X 0,Y 538.075,Z 190.768,A -85,B 0,C 180,E1 -3948.701,E2 -3948.701} C_VEL
LIN {X 0,Y 538.081,Z 190.774,A -85,B 0,C 180,E1 -3951.739,E2 -3951.739} C_VEL
LIN {X 0,Y 538.157,Z 190.758,A -85,B 0,C 180,E1 -3954.755,E2 -3954.755} C_VEL
LIN {X 0,Y 538.161,Z 190.766,A -85,B 0,C 180,E1 -3957.754,E2 -3957.754} C_VEL
LIN {X 0,Y 538.178,Z 190.755,A -85,B 0,C 180,E1 -3960.748,E2 -3960.748} C_VEL
LIN {X 0,Y 538.134,Z 190.762,A -85,B 0,C 180,E1 -3962.994,E2 -3962.994} C_VEL
LIN {X 0,Y 538.115,Z 190.766,A -85,B 0,C 180,E1 -3965.997,E2 -3965.997} C_VEL
LIN {X 0,Y 538.056,Z 190.772,A -85,B 0,C 180,E1 -3969.017,E2 -3969.017} C_VEL
LIN {X 0,Y 538.063,Z 190.771,A -85,B 0,C 180,E1 -3972.063,E2 -3972.063} C_VEL
LIN {X 0,Y 538.041,Z 190.777,A -85,B 0,C 180,E1 -3975.144,E2 -3975.144} C_VEL
LIN {X 0,Y 538.021,Z 190.774,A -85,B 0,C 180,E1 -3978.27,E2 -3978.27} C_VEL
LIN {X 0,Y 538.033,Z 190.774,A -85,B 0,C 180,E1 -3980.651,E2 -3980.651} C_VEL
LIN {X 0,Y 537.999,Z 190.778,A -85,B 0,C 180,E1 -3983.888,E2 -3983.888} C_VEL
LIN {X 0,Y 538.037,Z 190.772,A -85,B 0,C 180,E1 -3986.367,E2 -3986.367} C_VEL
LIN {X 0,Y 538.027,Z 190.779,A -85,B 0,C 180,E1 -3988.933,E2 -3988.933} C_VEL
LIN {X 0,Y 538.007,Z 190.776,A -85,B 0,C 180,E1 -3991.887,E2 -3991.887} C_VEL
LIN {X 0,Y 538.007,Z 190.778,A -85,B 0,C 180,E1 -3994.617,E2 -3994.617} C_VEL
LIN {X 0,Y 538.002,Z 190.786,A -85,B 0,C 180,E1 -3997.169,E2 -3997.169} C_VEL
LIN {X 0,Y 538.019,Z 190.776,A -85,B 0,C 180,E1 -3999.797,E2 -3999.797} C_VEL
LIN {X 0,Y 537.986,Z 190.785,A -85,B 0,C 180,E1 -4002.789,E2 -4002.789} C_VEL
LIN {X 0,Y 537.999,Z 190.785,A -85,B 0,C 180,E1 -4005.137,E2 -4005.137} C_VEL
LIN {X 0,Y 537.999,Z 190.778,A -85,B 0,C 180,E1 -4008.223,E2 -4008.223} C_VEL
LIN {X 0,Y 538.012,Z 190.782,A -85,B 0,C 180,E1 -4011.169,E2 -4011.169} C_VEL
LIN {X 0,Y 537.989,Z 190.781,A -85,B 0,C 180,E1 -4014.089,E2 -4014.089} C_VEL
LIN {X 0,Y 538.032,Z 190.781,A -85,B 0,C 180,E1 -4016.727,E2 -4016.727} C_VEL
LIN {X 0,Y 538.007,Z 190.782,A -85,B 0,C 180,E1 -4019.559,E2 -4019.559} C_VEL
LIN {X 0,Y 538.027,Z 190.965,A -85,B 0,C 180,E1 -4020.521,E2 -4020.521} C_VEL
LIN {X 0,Y 541.937,Z 204.046,A -85,B 0,C 180,E1 -4021.986,E2 -4021.986} C_VEL
LIN {X 0,Y 542.231,Z 207.119,A -85,B 0,C 180,E1 -4022.29,E2 -4022.29} C_VEL
LIN {X 0,Y 541.484,Z 234.081,A -85,B 0,C 180,E1 -4024.764,E2 -4024.764} C_VEL
LIN {X 0,Y 543.768,Z 247.565,A -85,B 0,C 180,E1 -4025.078,E2 -4025.078} C_VEL
LIN {X 0,Y 542.451,Z 439.858,A -85,B 0,C 180,E1 -4027.755,E2 -4027.755} C_VEL
LIN {X 0,Y 542.207,Z 456.369,A -85,B 0,C 180,E1 -4028.12,E2 -4028.12} C_VEL
LIN {X 0,Y 541.779,Z 473.293,A -85,B 0,C 180,E1 -4028.651,E2 -4028.651} C_VEL
LIN {X 0,Y 541.398,Z 488.627,A -85,B 0,C 180,E1 -4029.285,E2 -4029.285} C_VEL
LIN {X 0,Y 540.84,Z 503.623,A -85,B 0,C 180,E1 -4030.054,E2 -4030.054} C_VEL
LIN {X 0,Y 540.297,Z 518.971,A -85,B 0,C 180,E1 -4031.022,E2 -4031.022} C_VEL
LIN {X 0,Y 539.81,Z 532.053,A -85,B 0,C 180,E1 -4032.004,E2 -4032.004} C_VEL
LIN {X 0,Y 539.344,Z 545.032,A -85,B 0,C 180,E1 -4033.145,E2 -4033.145} C_VEL
LIN {X 0,Y 538.951,Z 556.271,A -85,B 0,C 180,E1 -4034.3,E2 -4034.3} C_VEL
LIN {X 0,Y 538.575,Z 567.409,A -85,B 0,C 180,E1 -4035.643,E2 -4035.643} C_VEL
LIN {X 0,Y 538.206,Z 578.197,A -85,B 0,C 180,E1 -4037.173,E2 -4037.173} C_VEL
LIN {X 0,Y 537.992,Z 587.259,A -85,B 0,C 180,E1 -4038.698,E2 -4038.698} C_VEL
LIN {X 0,Y 537.74,Z 594.848,A -85,B 0,C 180,E1 -4040.216,E2 -4040.216} C_VEL
LIN {X 0,Y 537.66,Z 602.459,A -85,B 0,C 180,E1 -4042.11,E2 -4042.11} C_VEL
LIN {X 0,Y 537.588,Z 608.245,A -85,B 0,C 180,E1 -4043.995,E2 -4043.995} C_VEL
LIN {X 0,Y 537.5,Z 611.631,A -85,B 0,C 180,E1 -4045.499,E2 -4045.499} C_VEL
LIN {X 0,Y 537.539,Z 614.088,A -85,B 0,C 180,E1 -4047.001,E2 -4047.001} C_VEL
LIN {X 0,Y 537.445,Z 615.477,A -85,B 0,C 180,E1 -4048.5,E2 -4048.5} C_VEL
LIN {X 0,Y 537.437,Z 616,A -85,B 0,C 180,E1 -4049.998,E2 -4049.998} C_VEL
LIN {X 0,Y 537.445,Z 615.479,A -85,B 0,C 180,E1 -4051.497,E2 -4051.497} C_VEL
LIN {X 0,Y 537.538,Z 614.092,A -85,B 0,C 180,E1 -4052.996,E2 -4052.996} C_VEL
LIN {X 0,Y 537.499,Z 611.637,A -85,B 0,C 180,E1 -4054.498,E2 -4054.498} C_VEL
LIN {X 0,Y 537.586,Z 608.258,A -85,B 0,C 180,E1 -4056.001,E2 -4056.001} C_VEL
LIN {X 0,Y 537.659,Z 602.475,A -85,B 0,C 180,E1 -4057.887,E2 -4057.887} C_VEL
LIN {X 0,Y 537.741,Z 594.866,A -85,B 0,C 180,E1 -4059.78,E2 -4059.78} C_VEL
LIN {X 0,Y 537.986,Z 587.279,A -85,B 0,C 180,E1 -4061.298,E2 -4061.298} C_VEL
LIN {X 0,Y 538.202,Z 578.222,A -85,B 0,C 180,E1 -4062.824,E2 -4062.824} C_VEL
LIN {X 0,Y 538.583,Z 567.438,A -85,B 0,C 180,E1 -4064.353,E2 -4064.353} C_VEL
LIN {X 0,Y 538.972,Z 556.306,A -85,B 0,C 180,E1 -4065.696,E2 -4065.696} C_VEL
LIN {X 0,Y 539.391,Z 544.092,A -85,B 0,C 180,E1 -4066.947,E2 -4066.947} C_VEL
LIN {X 0,Y 539.955,Z 529.954,A -85,B 0,C 180,E1 -4068.166,E2 -4068.166} C_VEL
LIN {X 0,Y 540.431,Z 516.185,A -85,B 0,C 180,E1 -4069.167,E2 -4069.167} C_VEL
LIN {X 0,Y 540.882,Z 501.953,A -85,B 0,C 180,E1 -4070.039,E2 -4070.039} C_VEL
LIN {X 0,Y 541.441,Z 486.586,A -85,B 0,C 180,E1 -4070.812,E2 -4070.812} C_VEL
LIN {X 0,Y 541.911,Z 470.863,A -85,B 0,C 180,E1 -4071.439,E2 -4071.439} C_VEL
LIN {X 0,Y 542.216,Z 454.771,A -85,B 0,C 180,E1 -4071.926,E2 -4071.926} C_VEL
LIN {X 0,Y 542.514,Z 438.714,A -85,B 0,C 180,E1 -4072.264,E2 -4072.264} C_VEL
LIN {X 0,Y 543.743,Z 246.672,A -85,B 0,C 180,E1 -4074.938,E2 -4074.938} C_VEL
LIN {X 0,Y 541.517,Z 234.028,A -85,B 0,C 180,E1 -4075.255,E2 -4075.255} C_VEL
LIN {X 0,Y 542.33,Z 206.233,A -85,B 0,C 180,E1 -4077.805,E2 -4077.805} C_VEL
LIN {X 0,Y 540.224,Z 198.349,A -85,B 0,C 180,E1 -4078.668,E2 -4078.668} C_VEL
LIN {X 0,Y 538.011,Z 190.784,A -85,B 0,C 180,E1 -4079.53,E2 -4079.53} C_VEL
LIN {X 0,Y 538.01,Z 190.774,A -85,B 0,C 180,E1 -4082.38,E2 -4082.38} C_VEL
LIN {X 0,Y 537.988,Z 190.787,A -85,B 0,C 180,E1 -4085.081,E2 -4085.081} C_VEL
LIN {X 0,Y 537.972,Z 190.783,A -85,B 0,C 180,E1 -4087.875,E2 -4087.875} C_VEL
LIN {X 0,Y 538.029,Z 190.776,A -85,B 0,C 180,E1 -4090.773,E2 -4090.773} C_VEL
LIN {X 0,Y 538.001,Z 190.778,A -85,B 0,C 180,E1 -4094.072,E2 -4094.072} C_VEL
LIN {X 0,Y 538.002,Z 190.783,A -85,B 0,C 180,E1 -4097.01,E2 -4097.01} C_VEL
LIN {X 0,Y 538.052,Z 190.775,A -85,B 0,C 180,E1 -4099.247,E2 -4099.247} C_VEL
LIN {X 0,Y 537.967,Z 190.781,A -85,B 0,C 180,E1 -4102.121,E2 -4102.121} C_VEL
LIN {X 0,Y 537.991,Z 190.783,A -85,B 0,C 180,E1 -4104.915,E2 -4104.915} C_VEL
LIN {X 0,Y 538.001,Z 190.773,A -85,B 0,C 180,E1 -4107.616,E2 -4107.616} C_VEL
LIN {X 0,Y 537.988,Z 190.779,A -85,B 0,C 180,E1 -4110.237,E2 -4110.237} C_VEL
LIN {X 0,Y 538.036,Z 190.779,A -85,B 0,C 180,E1 -4112.795,E2 -4112.795} C_VEL
LIN {X 0,Y 538.02,Z 190.779,A -85,B 0,C 180,E1 -4115.292,E2 -4115.292} C_VEL
LIN {X 0,Y 538.014,Z 190.775,A -85,B 0,C 180,E1 -4118.032,E2 -4118.032} C_VEL
LIN {X 0,Y 538.01,Z 190.778,A -85,B 0,C 180,E1 -4120.939,E2 -4120.939} C_VEL
LIN {X 0,Y 537.994,Z 190.781,A -85,B 0,C 180,E1 -4123.298,E2 -4123.298} C_VEL
LIN {X 0,Y 538.03,Z 190.771,A -85,B 0,C 180,E1 -4125.63,E2 -4125.63} C_VEL
LIN {X 0,Y 538.074,Z 190.765,A -85,B 0,C 180,E1 -4128.702,E2 -4128.702} C_VEL
LIN {X 0,Y 538.055,Z 190.77,A -85,B 0,C 180,E1 -4131.739,E2 -4131.739} C_VEL
LIN {X 0,Y 538.153,Z 190.759,A -85,B 0,C 180,E1 -4134.755,E2 -4134.755} C_VEL
LIN {X 0,Y 538.129,Z 190.755,A -85,B 0,C 180,E1 -4137.755,E2 -4137.755} C_VEL
LIN {X 0,Y 538.158,Z 190.766,A -85,B 0,C 180,E1 -4140.749,E2 -4140.749} C_VEL
LIN {X 0,Y 538.112,Z 190.763,A -85,B 0,C 180,E1 -4142.995,E2 -4142.995} C_VEL
LIN {X 0,Y 538.089,Z 190.764,A -85,B 0,C 180,E1 -4145.998,E2 -4145.998} C_VEL
LIN {X 0,Y 538.045,Z 190.773,A -85,B 0,C 180,E1 -4149.018,E2 -4149.018} C_VEL
LIN {X 0,Y 538.051,Z 190.766,A -85,B 0,C 180,E1 -4152.064,E2 -4152.064} C_VEL
LIN {X 0,Y 538.014,Z 190.776,A -85,B 0,C 180,E1 -4155.145,E2 -4155.145} C_VEL
LIN {X 0,Y 538.032,Z 190.77,A -85,B 0,C 180,E1 -4157.544,E2 -4157.544} C_VEL
LIN {X 0,Y 538.014,Z 190.781,A -85,B 0,C 180,E1 -4160.653,E2 -4160.653} C_VEL
LIN {X 0,Y 538.012,Z 190.777,A -85,B 0,C 180,E1 -4163.888,E2 -4163.888} C_VEL
LIN {X 0,Y 538.013,Z 190.777,A -85,B 0,C 180,E1 -4166.369,E2 -4166.369} C_VEL
LIN {X 0,Y 538.005,Z 190.778,A -85,B 0,C 180,E1 -4168.936,E2 -4168.936} C_VEL
LIN {X 0,Y 537.984,Z 190.78,A -85,B 0,C 180,E1 -4171.89,E2 -4171.89} C_VEL
LIN {X 0,Y 538.001,Z 190.781,A -85,B 0,C 180,E1 -4174.622,E2 -4174.622} C_VEL
LIN {X 0,Y 537.982,Z 190.778,A -85,B 0,C 180,E1 -4177.173,E2 -4177.173} C_VEL
LIN {X 0,Y 537.99,Z 190.775,A -85,B 0,C 180,E1 -4179.8,E2 -4179.8} C_VEL
LIN {X 0,Y 537.992,Z 190.775,A -85,B 0,C 180,E1 -4180.296,E2 -4180.296} C_VEL
LIN {X 0,Y 537.351,Z 190.86,A -85,B 0,C 180,E1 -4180.922,E2 -4180.922} C_VEL
LIN {X 0,Y 534.499,Z 191.217,A -85,B 0,C 180,E1 -4181.937,E2 -4181.937} C_VEL
LIN {X 0,Y 532.068,Z 191.519,A -85,B 0,C 180,E1 -4182.754,E2 -4182.754} C_VEL
LIN {X 0,Y 531.018,Z 191.647,A -85,B 0,C 180,E1 -4183.385,E2 -4183.385} C_VEL
LIN {X 0,Y 530.93,Z 191.657,A -85,B 0,C 180,E1 -4183.599,E2 -4183.599} C_VEL
LIN {X 0,Y 530.926,Z 191.663,A -85,B 0,C 180,E1 -4186.506,E2 -4186.506} C_VEL
LIN {X 0,Y 530.964,Z 191.654,A -85,B 0,C 180,E1 -4189.57,E2 -4189.57} C_VEL
LIN {X 0,Y 530.954,Z 191.658,A -85,B 0,C 180,E1 -4192.58,E2 -4192.58} C_VEL
LIN {X 0,Y 530.975,Z 191.649,A -85,B 0,C 180,E1 -4195.313,E2 -4195.313} C_VEL
LIN {X 0,Y 530.956,Z 191.663,A -85,B 0,C 180,E1 -4198.035,E2 -4198.035} C_VEL
LIN {X 0,Y 530.979,Z 191.651,A -85,B 0,C 180,E1 -4200.877,E2 -4200.877} C_VEL
LIN {X 0,Y 530.961,Z 191.659,A -85,B 0,C 180,E1 -4204.103,E2 -4204.103} C_VEL
LIN {X 0,Y 530.944,Z 191.657,A -85,B 0,C 180,E1 -4206.606,E2 -4206.606} C_VEL
LIN {X 0,Y 530.987,Z 191.652,A -85,B 0,C 180,E1 -4209.064,E2 -4209.064} C_VEL
LIN {X 0,Y 530.962,Z 191.656,A -85,B 0,C 180,E1 -4211.48,E2 -4211.48} C_VEL
LIN {X 0,Y 530.981,Z 191.653,A -85,B 0,C 180,E1 -4214.652,E2 -4214.652} C_VEL
LIN {X 0,Y 531.022,Z 191.655,A -85,B 0,C 180,E1 -4217.777,E2 -4217.777} C_VEL
LIN {X 0,Y 530.972,Z 191.658,A -85,B 0,C 180,E1 -4220.094,E2 -4220.094} C_VEL
LIN {X 0,Y 531.015,Z 191.65,A -85,B 0,C 180,E1 -4223.161,E2 -4223.161} C_VEL
LIN {X 0,Y 530.985,Z 191.653,A -85,B 0,C 180,E1 -4225.447,E2 -4225.447} C_VEL
LIN {X 0,Y 531.137,Z 191.64,A -85,B 0,C 180,E1 -4227.727,E2 -4227.727} C_VEL
LIN {X 0,Y 531.089,Z 191.841,A -85,B 0,C 180,E1 -4229.646,E2 -4229.646} C_VEL
LIN {X 0,Y 534.712,Z 205.293,A -85,B 0,C 180,E1 -4231.32,E2 -4231.32} C_VEL
LIN {X 0,Y 534.795,Z 207.179,A -85,B 0,C 180,E1 -4231.496,E2 -4231.496} C_VEL
LIN {X 0,Y 537.382,Z 220.179,A -85,B 0,C 180,E1 -4231.819,E2 -4231.819} C_VEL
LIN {X 0,Y 535.941,Z 412.19,A -85,B 0,C 180,E1 -4234.538,E2 -4234.538} C_VEL
LIN {X 0,Y 535.618,Z 429.59,A -85,B 0,C 180,E1 -4234.941,E2 -4234.941} C_VEL
LIN {X 0,Y 535.187,Z 445.471,A -85,B 0,C 180,E1 -4235.465,E2 -4235.465} C_VEL
LIN {X 0,Y 534.728,Z 460.976,A -85,B 0,C 180,E1 -4236.132,E2 -4236.132} C_VEL
LIN {X 0,Y 534.143,Z 476.92,A -85,B 0,C 180,E1 -4236.992,E2 -4236.992} C_VEL
LIN {X 0,Y 533.554,Z 491.433,A -85,B 0,C 180,E1 -4237.951,E2 -4237.951} C_VEL
LIN {X 0,Y 532.987,Z 504.663,A -85,B 0,C 180,E1 -4238.991,E2 -4238.991} C_VEL
LIN {X 0,Y 532.469,Z 516.47,A -85,B 0,C 180,E1 -4240.073,E2 -4240.073} C_VEL
LIN {X 0,Y 531.943,Z 529.087,A -85,B 0,C 180,E1 -4241.432,E2 -4241.432} C_VEL
LIN {X 0,Y 531.505,Z 539.819,A -85,B 0,C 180,E1 -4242.797,E2 -4242.797} C_VEL
LIN {X 0,Y 531.188,Z 549.062,A -85,B 0,C 180,E1 -4244.169,E2 -4244.169} C_VEL
LIN {X 0,Y 530.911,Z 558.097,A -85,B 0,C 180,E1 -4245.747,E2 -4245.747} C_VEL
LIN {X 0,Y 530.703,Z 565.303,A -85,B 0,C 180,E1 -4247.235,E2 -4247.235} C_VEL
LIN {X 0,Y 530.59,Z 572.037,A -85,B 0,C 180,E1 -4248.938,E2 -4248.938} C_VEL
LIN {X 0,Y 530.514,Z 577.118,A -85,B 0,C 180,E1 -4250.553,E2 -4250.553} C_VEL
LIN {X 0,Y 530.391,Z 580.565,A -85,B 0,C 180,E1 -4251.944,E2 -4251.944} C_VEL
LIN {X 0,Y 530.34,Z 583.905,A -85,B 0,C 180,E1 -4253.881,E2 -4253.881} C_VEL
LIN {X 0,Y 530.352,Z 585.583,A -85,B 0,C 180,E1 -4255.695,E2 -4255.695} C_VEL
LIN {X 0,Y 530.374,Z 585.933,A -85,B 0,C 180,E1 -4257.399,E2 -4257.399} C_VEL
LIN {X 0,Y 530.389,Z 585.202,A -85,B 0,C 180,E1 -4259.008,E2 -4259.008} C_VEL
LIN {X 0,Y 530.39,Z 583.429,A -85,B 0,C 180,E1 -4260.537,E2 -4260.537} C_VEL
LIN {X 0,Y 530.386,Z 580.874,A -85,B 0,C 180,E1 -4262.008,E2 -4262.008} C_VEL
LIN {X 0,Y 530.493,Z 576.368,A -85,B 0,C 180,E1 -4263.809,E2 -4263.809} C_VEL
LIN {X 0,Y 530.617,Z 570.23,A -85,B 0,C 180,E1 -4265.647,E2 -4265.647} C_VEL
LIN {X 0,Y 530.777,Z 562.809,A -85,B 0,C 180,E1 -4267.395,E2 -4267.395} C_VEL
LIN {X 0,Y 531.037,Z 554.458,A -85,B 0,C 180,E1 -4269.011,E2 -4269.011} C_VEL
LIN {X 0,Y 531.316,Z 544.364,A -85,B 0,C 180,E1 -4270.645,E2 -4270.645} C_VEL
LIN {X 0,Y 531.729,Z 533.901,A -85,B 0,C 180,E1 -4272.072,E2 -4272.072} C_VEL
LIN {X 0,Y 532.254,Z 522.22,A -85,B 0,C 180,E1 -4273.428,E2 -4273.428} C_VEL
LIN {X 0,Y 532.771,Z 509.412,A -85,B 0,C 180,E1 -4274.688,E2 -4274.688} C_VEL
LIN {X 0,Y 533.339,Z 496.246,A -85,B 0,C 180,E1 -4275.785,E2 -4275.785} C_VEL
LIN {X 0,Y 533.974,Z 481.578,A -85,B 0,C 180,E1 -4276.81,E2 -4276.81} C_VEL
LIN {X 0,Y 534.472,Z 467.684,A -85,B 0,C 180,E1 -4277.622,E2 -4277.622} C_VEL
LIN {X 0,Y 535.046,Z 451.511,A -85,B 0,C 180,E1 -4278.386,E2 -4278.386} C_VEL
LIN {X 0,Y 535.497,Z 434.553,A -85,B 0,C 180,E1 -4279.003,E2 -4279.003} C_VEL
LIN {X 0,Y 535.87,Z 418.416,A -85,B 0,C 180,E1 -4279.426,E2 -4279.426} C_VEL
LIN {X 0,Y 536.077,Z 400.695,A -85,B 0,C 180,E1 -4279.731,E2 -4279.731} C_VEL
LIN {X 0,Y 537.386,Z 219.259,A -85,B 0,C 180,E1 -4282.287,E2 -4282.287} C_VEL
LIN {X 0,Y 534.825,Z 206.952,A -85,B 0,C 180,E1 -4282.61,E2 -4282.61} C_VEL
LIN {X 0,Y 534.329,Z 203.56,A -85,B 0,C 180,E1 -4283.005,E2 -4283.005} C_VEL
LIN {X 0,Y 530.99,Z 191.659,A -85,B 0,C 180,E1 -4284.513,E2 -4284.513} C_VEL
LIN {X 0,Y 530.969,Z 191.657,A -85,B 0,C 180,E1 -4287.133,E2 -4287.133} C_VEL
LIN {X 0,Y 530.971,Z 191.658,A -85,B 0,C 180,E1 -4289.803,E2 -4289.803} C_VEL
LIN {X 0,Y 531.016,Z 191.654,A -85,B 0,C 180,E1 -4292.467,E2 -4292.467} C_VEL
LIN {X 0,Y 530.995,Z 191.653,A -85,B 0,C 180,E1 -4294.941,E2 -4294.941} C_VEL
LIN {X 0,Y 530.971,Z 191.658,A -85,B 0,C 180,E1 -4298.246,E2 -4298.246} C_VEL
LIN {X 0,Y 530.995,Z 191.653,A -85,B 0,C 180,E1 -4300.677,E2 -4300.677} C_VEL
LIN {X 0,Y 530.985,Z 191.649,A -85,B 0,C 180,E1 -4303.071,E2 -4303.071} C_VEL
LIN {X 0,Y 531.018,Z 191.649,A -85,B 0,C 180,E1 -4305.435,E2 -4305.435} C_VEL
LIN {X 0,Y 531.035,Z 191.646,A -85,B 0,C 180,E1 -4308.549,E2 -4308.549} C_VEL
LIN {X 0,Y 531.05,Z 191.649,A -85,B 0,C 180,E1 -4311.629,E2 -4311.629} C_VEL
LIN {X 0,Y 531.116,Z 191.635,A -85,B 0,C 180,E1 -4314.685,E2 -4314.685} C_VEL
LIN {X 0,Y 531.133,Z 191.641,A -85,B 0,C 180,E1 -4317.725,E2 -4317.725} C_VEL
LIN {X 0,Y 531.149,Z 191.631,A -85,B 0,C 180,E1 -4320.758,E2 -4320.758} C_VEL
LIN {X 0,Y 531.101,Z 191.638,A -85,B 0,C 180,E1 -4323.034,E2 -4323.034} C_VEL
LIN {X 0,Y 531.071,Z 191.643,A -85,B 0,C 180,E1 -4326.077,E2 -4326.077} C_VEL
LIN {X 0,Y 531.018,Z 191.65,A -85,B 0,C 180,E1 -4329.138,E2 -4329.138} C_VEL
LIN {X 0,Y 531.026,Z 191.646,A -85,B 0,C 180,E1 -4332.225,E2 -4332.225} C_VEL
LIN {X 0,Y 530.991,Z 191.658,A -85,B 0,C 180,E1 -4335.349,E2 -4335.349} C_VEL
LIN {X 0,Y 530.981,Z 191.651,A -85,B 0,C 180,E1 -4338.521,E2 -4338.521} C_VEL
LIN {X 0,Y 530.995,Z 191.653,A -85,B 0,C 180,E1 -4340.938,E2 -4340.938} C_VEL
LIN {X 0,Y 530.961,Z 191.653,A -85,B 0,C 180,E1 -4344.225,E2 -4344.225} C_VEL
LIN {X 0,Y 530.998,Z 191.652,A -85,B 0,C 180,E1 -4346.744,E2 -4346.744} C_VEL
LIN {X 0,Y 530.977,Z 191.658,A -85,B 0,C 180,E1 -4349.322,E2 -4349.322} C_VEL
LIN {X 0,Y 530.962,Z 191.653,A -85,B 0,C 180,E1 -4352.1,E2 -4352.1} C_VEL
LIN {X 0,Y 530.966,Z 191.658,A -85,B 0,C 180,E1 -4354.85,E2 -4354.85} C_VEL
LIN {X 0,Y 530.963,Z 191.657,A -85,B 0,C 180,E1 -4357.507,E2 -4357.507} C_VEL
LIN {X 0,Y 530.979,Z 191.654,A -85,B 0,C 180,E1 -4360.433,E2 -4360.433} C_VEL
LIN {X 0,Y 530.932,Z 191.663,A -85,B 0,C 180,E1 -4363.277,E2 -4363.277} C_VEL
LIN {X 0,Y 530.974,Z 191.656,A -85,B 0,C 180,E1 -4365.622,E2 -4365.622} C_VEL
LIN {X 0,Y 530.962,Z 191.658,A -85,B 0,C 180,E1 -4368.561,E2 -4368.561} C_VEL
LIN {X 0,Y 530.955,Z 191.658,A -85,B 0,C 180,E1 -4371.529,E2 -4371.529} C_VEL
LIN {X 0,Y 530.95,Z 191.661,A -85,B 0,C 180,E1 -4374.379,E2 -4374.379} C_VEL
LIN {X 0,Y 530.967,Z 191.659,A -85,B 0,C 180,E1 -4377.133,E2 -4377.133} C_VEL
LIN {X 0,Y 530.971,Z 191.731,A -85,B 0,C 180,E1 -4380.186,E2 -4380.186} C_VEL
LIN {X 0,Y 535.622,Z 208.004,A -85,B 0,C 180,E1 -4382.024,E2 -4382.024} C_VEL
LIN {X 0,Y 534.809,Z 233.939,A -85,B 0,C 180,E1 -4384.435,E2 -4384.435} C_VEL
LIN {X 0,Y 537.306,Z 247.683,A -85,B 0,C 180,E1 -4384.762,E2 -4384.762} C_VEL
LIN {X 0,Y 535.869,Z 440.915,A -85,B 0,C 180,E1 -4387.492,E2 -4387.492} C_VEL
LIN {X 0,Y 535.57,Z 456.924,A -85,B 0,C 180,E1 -4387.86,E2 -4387.86} C_VEL
LIN {X 0,Y 535.13,Z 472.969,A -85,B 0,C 180,E1 -4388.373,E2 -4388.373} C_VEL
LIN {X 0,Y 534.712,Z 487.975,A -85,B 0,C 180,E1 -4388.996,E2 -4388.996} C_VEL
LIN {X 0,Y 534.079,Z 503.331,A -85,B 0,C 180,E1 -4389.791,E2 -4389.791} C_VEL
LIN {X 0,Y 533.526,Z 518.695,A -85,B 0,C 180,E1 -4390.771,E2 -4390.771} C_VEL
LIN {X 0,Y 532.916,Z 532.617,A -85,B 0,C 180,E1 -4391.833,E2 -4391.833} C_VEL
LIN {X 0,Y 532.459,Z 544.776,A -85,B 0,C 180,E1 -4392.92,E2 -4392.92} C_VEL
LIN {X 0,Y 532.011,Z 556.046,A -85,B 0,C 180,E1 -4394.09,E2 -4394.09} C_VEL
LIN {X 0,Y 531.6,Z 567.29,A -85,B 0,C 180,E1 -4395.451,E2 -4395.451} C_VEL
LIN {X 0,Y 531.193,Z 578.18,A -85,B 0,C 180,E1 -4397,E2 -4397} C_VEL
LIN {X 0,Y 530.969,Z 587.259,A -85,B 0,C 180,E1 -4398.547,E2 -4398.547} C_VEL
LIN {X 0,Y 530.697,Z 594.848,A -85,B 0,C 180,E1 -4400.085,E2 -4400.085} C_VEL
LIN {X 0,Y 530.57,Z 602.459,A -85,B 0,C 180,E1 -4402.004,E2 -4402.004} C_VEL
LIN {X 0,Y 530.496,Z 608.245,A -85,B 0,C 180,E1 -4403.915,E2 -4403.915} C_VEL
LIN {X 0,Y 530.403,Z 611.63,A -85,B 0,C 180,E1 -4405.438,E2 -4405.438} C_VEL
LIN {X 0,Y 530.444,Z 614.089,A -85,B 0,C 180,E1 -4406.96,E2 -4406.96} C_VEL
LIN {X 0,Y 530.355,Z 615.477,A -85,B 0,C 180,E1 -4408.48,E2 -4408.48} C_VEL
LIN {X 0,Y 530.338,Z 616,A -85,B 0,C 180,E1 -4409.998,E2 -4409.998} C_VEL
LIN {X 0,Y 530.355,Z 615.478,A -85,B 0,C 180,E1 -4411.517,E2 -4411.517} C_VEL
LIN {X 0,Y 530.443,Z 614.092,A -85,B 0,C 180,E1 -4413.036,E2 -4413.036} C_VEL
LIN {X 0,Y 530.402,Z 611.637,A -85,B 0,C 180,E1 -4414.558,E2 -4414.558} C_VEL
LIN {X 0,Y 530.493,Z 608.258,A -85,B 0,C 180,E1 -4416.082,E2 -4416.082} C_VEL
LIN {X 0,Y 530.57,Z 602.475,A -85,B 0,C 180,E1 -4417.993,E2 -4417.993} C_VEL
LIN {X 0,Y 530.696,Z 594.865,A -85,B 0,C 180,E1 -4419.911,E2 -4419.911} C_VEL
LIN {X 0,Y 530.996,Z 586.264,A -85,B 0,C 180,E1 -4421.644,E2 -4421.644} C_VEL
LIN {X 0,Y 531.225,Z 576.964,A -85,B 0,C 180,E1 -4423.19,E2 -4423.19} C_VEL
LIN {X 0,Y 531.606,Z 567.329,A -85,B 0,C 180,E1 -4424.545,E2 -4424.545} C_VEL
LIN {X 0,Y 532.027,Z 556.1,A -85,B 0,C 180,E1 -4425.906,E2 -4425.906} C_VEL
LIN {X 0,Y 532.526,Z 543.861,A -85,B 0,C 180,E1 -4427.173,E2 -4427.173} C_VEL
LIN {X 0,Y 533.074,Z 530.605,A -85,B 0,C 180,E1 -4428.334,E2 -4428.334} C_VEL
LIN {X 0,Y 533.575,Z 517.373,A -85,B 0,C 180,E1 -4429.323,E2 -4429.323} C_VEL
LIN {X 0,Y 534.08,Z 503.469,A -85,B 0,C 180,E1 -4430.205,E2 -4430.205} C_VEL
LIN {X 0,Y 534.695,Z 487.843,A -85,B 0,C 180,E1 -4431.016,E2 -4431.016} C_VEL
LIN {X 0,Y 535.19,Z 473.186,A -85,B 0,C 180,E1 -4431.621,E2 -4431.621} C_VEL
LIN {X 0,Y 535.549,Z 457.21,A -85,B 0,C 180,E1 -4432.137,E2 -4432.137} C_VEL
LIN {X 0,Y 535.886,Z 441.342,A -85,B 0,C 180,E1 -4432.503,E2 -4432.503} C_VEL
LIN {X 0,Y 537.313,Z 249.207,A -85,B 0,C 180,E1 -4435.218,E2 -4435.218} C_VEL
LIN {X 0,Y 536.712,Z 244.225,A -85,B 0,C 180,E1 -4435.321,E2 -4435.321} C_VEL
LIN {X 0,Y 534.846,Z 233.931,A -85,B 0,C 180,E1 -4435.583,E2 -4435.583} C_VEL
LIN {X 0,Y 535.688,Z 208.282,A -85,B 0,C 180,E1 -4437.968,E2 -4437.968} C_VEL
LIN {X 0,Y 532.189,Z 195.951,A -85,B 0,C 180,E1 -4439.357,E2 -4439.357} C_VEL
LIN {X 0,Y 530.964,Z 191.66,A -85,B 0,C 180,E1 -4439.865,E2 -4439.865} C_VEL
LIN {X 0,Y 530.953,Z 191.651,A -85,B 0,C 180,E1 -4442.864,E2 -4442.864} C_VEL
LIN {X 0,Y 530.939,Z 191.663,A -85,B 0,C 180,E1 -4445.617,E2 -4445.617} C_VEL
LIN {X 0,Y 530.947,Z 191.659,A -85,B 0,C 180,E1 -4448.651,E2 -4448.651} C_VEL
LIN {X 0,Y 530.974,Z 191.658,A -85,B 0,C 180,E1 -4451.433,E2 -4451.433} C_VEL
LIN {X 0,Y 530.963,Z 191.656,A -85,B 0,C 180,E1 -4454.545,E2 -4454.545} C_VEL
LIN {X 0,Y 530.963,Z 191.655,A -85,B 0,C 180,E1 -4457.831,E2 -4457.831} C_VEL
LIN {X 0,Y 530.964,Z 191.655,A -85,B 0,C 180,E1 -4460.555,E2 -4460.555} C_VEL
LIN {X 0,Y 530.945,Z 191.654,A -85,B 0,C 180,E1 -4463.841,E2 -4463.841} C_VEL
LIN {X 0,Y 530.97,Z 191.655,A -85,B 0,C 180,E1 -4466.492,E2 -4466.492} C_VEL
LIN {X 0,Y 530.944,Z 191.66,A -85,B 0,C 180,E1 -4469.353,E2 -4469.353} C_VEL
LIN {X 0,Y 530.985,Z 191.653,A -85,B 0,C 180,E1 -4472.465,E2 -4472.465} C_VEL
LIN {X 0,Y 530.975,Z 191.656,A -85,B 0,C 180,E1 -4474.941,E2 -4474.941} C_VEL
LIN {X 0,Y 530.975,Z 191.652,A -85,B 0,C 180,E1 -4477.889,E2 -4477.889} C_VEL
LIN {X 0,Y 530.966,Z 191.651,A -85,B 0,C 180,E1 -4480.677,E2 -4480.677} C_VEL
LIN {X 0,Y 530.959,Z 191.66,A -85,B 0,C 180,E1 -4483.071,E2 -4483.071} C_VEL
LIN {X 0,Y 530.985,Z 191.65,A -85,B 0,C 180,E1 -4485.435,E2 -4485.435} C_VEL
LIN {X 0,Y 531.026,Z 191.64,A -85,B 0,C 180,E1 -4488.55,E2 -4488.55} C_VEL
LIN {X 0,Y 531.024,Z 191.646,A -85,B 0,C 180,E1 -4491.629,E2 -4491.629} C_VEL
LIN {X 0,Y 531.108,Z 191.637,A -85,B 0,C 180,E1 -4494.686,E2 -4494.686} C_VEL
LIN {X 0,Y 531.102,Z 191.63,A -85,B 0,C 180,E1 -4497.725,E2 -4497.725} C_VEL
LIN {X 0,Y 531.127,Z 191.641,A -85,B 0,C 180,E1 -4500.759,E2 -4500.759} C_VEL
LIN {X 0,Y 531.078,Z 191.639,A -85,B 0,C 180,E1 -4503.035,E2 -4503.035} C_VEL
LIN {X 0,Y 531.049,Z 191.641,A -85,B 0,C 180,E1 -4506.078,E2 -4506.078} C_VEL
LIN {X 0,Y 531.004,Z 191.649,A -85,B 0,C 180,E1 -4509.139,E2 -4509.139} C_VEL
LIN {X 0,Y 531.008,Z 191.645,A -85,B 0,C 180,E1 -4512.226,E2 -4512.226} C_VEL
LIN {X 0,Y 530.966,Z 191.653,A -85,B 0,C 180,E1 -4515.351,E2 -4515.351} C_VEL
LIN {X 0,Y 530.987,Z 191.648,A -85,B 0,C 180,E1 -4517.724,E2 -4517.724} C_VEL
LIN {X 0,Y 530.975,Z 191.654,A -85,B 0,C 180,E1 -4520.939,E2 -4520.939} C_VEL
LIN {X 0,Y 530.978,Z 191.654,A -85,B 0,C 180,E1 -4524.047,E2 -4524.047} C_VEL
LIN {X 0,Y 530.977,Z 191.653,A -85,B 0,C 180,E1 -4526.746,E2 -4526.746} C_VEL
LIN {X 0,Y 530.955,Z 191.655,A -85,B 0,C 180,E1 -4529.325,E2 -4529.325} C_VEL
LIN {X 0,Y 530.939,Z 191.66,A -85,B 0,C 180,E1 -4532.103,E2 -4532.103} C_VEL
LIN {X 0,Y 530.958,Z 191.656,A -85,B 0,C 180,E1 -4534.856,E2 -4534.856} C_VEL
LIN {X 0,Y 530.943,Z 191.656,A -85,B 0,C 180,E1 -4537.51,E2 -4537.51} C_VEL
LIN {X 0,Y 530.958,Z 191.661,A -85,B 0,C 180,E1 -4540.436,E2 -4540.436} C_VEL
LIN {X 0,Y 530.94,Z 191.656,A -85,B 0,C 180,E1 -4543.284,E2 -4543.284} C_VEL
LIN {X 0,Y 530.93,Z 191.657,A -85,B 0,C 180,E1 -4543.599,E2 -4543.599} C_VEL
LIN {X 0,Y 530.258,Z 191.746,A -85,B 0,C 180,E1 -4544.233,E2 -4544.233} C_VEL
LIN {X 0,Y 527.402,Z 192.098,A -85,B 0,C 180,E1 -4545.262,E2 -4545.262} C_VEL
LIN {X 0,Y 524.995,Z 192.399,A -85,B 0,C 180,E1 -4546.09,E2 -4546.09} C_VEL
LIN {X 0,Y 523.964,Z 192.528,A -85,B 0,C 180,E1 -4546.73,E2 -4546.73} C_VEL
LIN {X 0,Y 523.881,Z 192.536,A -85,B 0,C 180,E1 -4546.946,E2 -4546.946} C_VEL
LIN {X 0,Y 523.933,Z 192.534,A -85,B 0,C 180,E1 -4549.923,E2 -4549.923} C_VEL
LIN {X 0,Y 523.896,Z 192.535,A -85,B 0,C 180,E1 -4552.871,E2 -4552.871} C_VEL
LIN {X 0,Y 523.923,Z 192.53,A -85,B 0,C 180,E1 -4555.713,E2 -4555.713} C_VEL
LIN {X 0,Y 523.909,Z 192.535,A -85,B 0,C 180,E1 -4558.459,E2 -4558.459} C_VEL
LIN {X 0,Y 523.917,Z 192.531,A -85,B 0,C 180,E1 -4561.127,E2 -4561.127} C_VEL
LIN {X 0,Y 523.91,Z 192.537,A -85,B 0,C 180,E1 -4563.998,E2 -4563.998} C_VEL
LIN {X 0,Y 523.902,Z 192.538,A -85,B 0,C 180,E1 -4566.272,E2 -4566.272} C_VEL
LIN {X 0,Y 523.936,Z 192.53,A -85,B 0,C 180,E1 -4568.769,E2 -4568.769} C_VEL
LIN {X 0,Y 523.925,Z 192.53,A -85,B 0,C 180,E1 -4571.223,E2 -4571.223} C_VEL
LIN {X 0,Y 523.878,Z 192.542,A -85,B 0,C 180,E1 -4573.64,E2 -4573.64} C_VEL
LIN {X 0,Y 523.921,Z 192.537,A -85,B 0,C 180,E1 -4576.03,E2 -4576.03} C_VEL
LIN {X 0,Y 523.991,Z 192.524,A -85,B 0,C 180,E1 -4579.179,E2 -4579.179} C_VEL
LIN {X 0,Y 523.955,Z 192.533,A -85,B 0,C 180,E1 -4581.517,E2 -4581.517} C_VEL
LIN {X 0,Y 524.035,Z 192.514,A -85,B 0,C 180,E1 -4584.615,E2 -4584.615} C_VEL
LIN {X 0,Y 524.107,Z 192.516,A -85,B 0,C 180,E1 -4587.696,E2 -4587.696} C_VEL
LIN {X 0,Y 523.932,Z 192.597,A -85,B 0,C 180,E1 -4589.305,E2 -4589.305} C_VEL
LIN {X 0,Y 528.043,Z 207.335,A -85,B 0,C 180,E1 -4591.145,E2 -4591.145} C_VEL
LIN {X 0,Y 530.966,Z 220.582,A -85,B 0,C 180,E1 -4591.496,E2 -4591.496} C_VEL
LIN {X 0,Y 529.382,Z 412.629,A -85,B 0,C 180,E1 -4594.251,E2 -4594.251} C_VEL
LIN {X 0,Y 529.034,Z 429.982,A -85,B 0,C 180,E1 -4594.66,E2 -4594.66} C_VEL
LIN {X 0,Y 528.578,Z 445.631,A -85,B 0,C 180,E1 -4595.184,E2 -4595.184} C_VEL
LIN {X 0,Y 528.098,Z 460.485,A -85,B 0,C 180,E1 -4595.826,E2 -4595.826} C_VEL
LIN {X 0,Y 527.457,Z 476.568,A -85,B 0,C 180,E1 -4596.697,E2 -4596.697} C_VEL
LIN {X 0,Y 526.788,Z 491.21,A -85,B 0,C 180,E1 -4597.668,E2 -4597.668} C_VEL
LIN {X 0,Y 526.203,Z 504.845,A -85,B 0,C 180,E1 -4598.752,E2 -4598.752} C_VEL
LIN {X 0,Y 525.553,Z 518.266,A -85,B 0,C 180,E1 -4600.013,E2 -4600.013} C_VEL
LIN {X 0,Y 524.978,Z 530.64,A -85,B 0,C 180,E1 -4601.39,E2 -4601.39} C_VEL
LIN {X 0,Y 524.493,Z 541.246,A -85,B 0,C 180,E1 -4602.775,E2 -4602.775} C_VEL
LIN {X 0,Y 524.116,Z 551.509,A -85,B 0,C 180,E1 -4604.365,E2 -4604.365} C_VEL
LIN {X 0,Y 523.818,Z 560.16,A -85,B 0,C 180,E1 -4605.966,E2 -4605.966} C_VEL
LIN {X 0,Y 523.605,Z 567.642,A -85,B 0,C 180,E1 -4607.637,E2 -4607.637} C_VEL
LIN {X 0,Y 523.499,Z 573.399,A -85,B 0,C 180,E1 -4609.204,E2 -4609.204} C_VEL
LIN {X 0,Y 523.391,Z 578.167,A -85,B 0,C 180,E1 -4610.846,E2 -4610.846} C_VEL
LIN {X 0,Y 523.305,Z 581.019,A -85,B 0,C 180,E1 -4612.09,E2 -4612.09} C_VEL
LIN {X 0,Y 523.255,Z 584.167,A -85,B 0,C 180,E1 -4614.029,E2 -4614.029} C_VEL
LIN {X 0,Y 523.25,Z 585.691,A -85,B 0,C 180,E1 -4615.853,E2 -4615.853} C_VEL
LIN {X 0,Y 523.27,Z 585.899,A -85,B 0,C 180,E1 -4617.57,E2 -4617.57} C_VEL
LIN {X 0,Y 523.299,Z 585.056,A -85,B 0,C 180,E1 -4619.194,E2 -4619.194} C_VEL
LIN {X 0,Y 523.311,Z 583.211,A -85,B 0,C 180,E1 -4620.737,E2 -4620.737} C_VEL
LIN {X 0,Y 523.348,Z 579.936,A -85,B 0,C 180,E1 -4622.491,E2 -4622.491} C_VEL
LIN {X 0,Y 523.417,Z 575.136,A -85,B 0,C 180,E1 -4624.329,E2 -4624.329} C_VEL
LIN {X 0,Y 523.549,Z 570.455,A -85,B 0,C 180,E1 -4625.728,E2 -4625.728} C_VEL
LIN {X 0,Y 523.715,Z 563.582,A -85,B 0,C 180,E1 -4627.402,E2 -4627.402} C_VEL
LIN {X 0,Y 524.006,Z 555.191,A -85,B 0,C 180,E1 -4629.078,E2 -4629.078} C_VEL
LIN {X 0,Y 524.299,Z 546.301,A -85,B 0,C 180,E1 -4630.57,E2 -4630.57} C_VEL
LIN {X 0,Y 524.71,Z 535.906,A -85,B 0,C 180,E1 -4632.045,E2 -4632.045} C_VEL
LIN {X 0,Y 525.288,Z 524.531,A -85,B 0,C 180,E1 -4633.412,E2 -4633.412} C_VEL
LIN {X 0,Y 525.873,Z 511.574,A -85,B 0,C 180,E1 -4634.738,E2 -4634.738} C_VEL
LIN {X 0,Y 526.538,Z 497.389,A -85,B 0,C 180,E1 -4635.958,E2 -4635.958} C_VEL
LIN {X 0,Y 527.175,Z 483.145,A -85,B 0,C 180,E1 -4636.983,E2 -4636.983} C_VEL
LIN {X 0,Y 527.832,Z 467.708,A -85,B 0,C 180,E1 -4637.9,E2 -4637.9} C_VEL
LIN {X 0,Y 528.419,Z 451.82,A -85,B 0,C 180,E1 -4638.659,E2 -4638.659} C_VEL
LIN {X 0,Y 528.895,Z 435.441,A -85,B 0,C 180,E1 -4639.264,E2 -4639.264} C_VEL
LIN {X 0,Y 529.308,Z 419.547,A -85,B 0,C 180,E1 -4639.694,E2 -4639.694} C_VEL
LIN {X 0,Y 529.524,Z 401.955,A -85,B 0,C 180,E1 -4640.009,E2 -4640.009} C_VEL
LIN {X 0,Y 530.917,Z 220.096,A -85,B 0,C 180,E1 -4642.607,E2 -4642.607} C_VEL
LIN {X 0,Y 528.046,Z 207.199,A -85,B 0,C 180,E1 -4642.962,E2 -4642.962} C_VEL
LIN {X 0,Y 523.954,Z 192.534,A -85,B 0,C 180,E1 -4644.851,E2 -4644.851} C_VEL
LIN {X 0,Y 523.937,Z 192.535,A -85,B 0,C 180,E1 -4647.679,E2 -4647.679} C_VEL
LIN {X 0,Y 523.955,Z 192.531,A -85,B 0,C 180,E1 -4650.676,E2 -4650.676} C_VEL
LIN {X 0,Y 523.975,Z 192.529,A -85,B 0,C 180,E1 -4653.728,E2 -4653.728} C_VEL
LIN {X 0,Y 523.914,Z 192.538,A -85,B 0,C 180,E1 -4656.269,E2 -4656.269} C_VEL
LIN {X 0,Y 523.946,Z 192.528,A -85,B 0,C 180,E1 -4658.766,E2 -4658.766} C_VEL
LIN {X 0,Y 523.952,Z 192.529,A -85,B 0,C 180,E1 -4661.22,E2 -4661.22} C_VEL
LIN {X 0,Y 523.935,Z 192.531,A -85,B 0,C 180,E1 -4663.638,E2 -4663.638} C_VEL
LIN {X 0,Y 523.938,Z 192.537,A -85,B 0,C 180,E1 -4666.028,E2 -4666.028} C_VEL
LIN {X 0,Y 524.012,Z 192.523,A -85,B 0,C 180,E1 -4668.394,E2 -4668.394} C_VEL
LIN {X 0,Y 523.998,Z 192.526,A -85,B 0,C 180,E1 -4671.515,E2 -4671.515} C_VEL
LIN {X 0,Y 524.078,Z 192.512,A -85,B 0,C 180,E1 -4674.613,E2 -4674.613} C_VEL
LIN {X 0,Y 524.106,Z 192.516,A -85,B 0,C 180,E1 -4677.694,E2 -4677.694} C_VEL
LIN {X 0,Y 524.119,Z 192.507,A -85,B 0,C 180,E1 -4680.768,E2 -4680.768} C_VEL
LIN {X 0,Y 524.067,Z 192.515,A -85,B 0,C 180,E1 -4683.075,E2 -4683.075} C_VEL
LIN {X 0,Y 524.033,Z 192.519,A -85,B 0,C 180,E1 -4686.159,E2 -4686.159} C_VEL
LIN {X 0,Y 523.988,Z 192.528,A -85,B 0,C 180,E1 -4689.262,E2 -4689.262} C_VEL
LIN {X 0,Y 523.996,Z 192.527,A -85,B 0,C 180,E1 -4691.737,E2 -4691.737} C_VEL
LIN {X 0,Y 523.99,Z 192.526,A -85,B 0,C 180,E1 -4695.052,E2 -4695.052} C_VEL
LIN {X 0,Y 523.944,Z 192.53,A -85,B 0,C 180,E1 -4697.969,E2 -4697.969} C_VEL
LIN {X 0,Y 523.955,Z 192.527,A -85,B 0,C 180,E1 -4700.41,E2 -4700.41} C_VEL
LIN {X 0,Y 523.908,Z 192.535,A -85,B 0,C 180,E1 -4702.893,E2 -4702.893} C_VEL
LIN {X 0,Y 523.98,Z 192.524,A -85,B 0,C 180,E1 -4706.019,E2 -4706.019} C_VEL
LIN {X 0,Y 523.927,Z 192.535,A -85,B 0,C 180,E1 -4708.875,E2 -4708.875} C_VEL
LIN {X 0,Y 523.917,Z 192.535,A -85,B 0,C 180,E1 -4711.544,E2 -4711.544} C_VEL
LIN {X 0,Y 523.918,Z 192.531,A -85,B 0,C 180,E1 -4714.291,E2 -4714.291} C_VEL
LIN {X 0,Y 523.905,Z 192.541,A -85,B 0,C 180,E1 -4717.132,E2 -4717.132} C_VEL
LIN {X 0,Y 523.937,Z 192.53,A -85,B 0,C 180,E1 -4720.129,E2 -4720.129} C_VEL
LIN {X 0,Y 523.917,Z 192.533,A -85,B 0,C 180,E1 -4722.456,E2 -4722.456} C_VEL
LIN {X 0,Y 523.939,Z 192.536,A -85,B 0,C 180,E1 -4725.31,E2 -4725.31} C_VEL
LIN {X 0,Y 523.923,Z 192.537,A -85,B 0,C 180,E1 -4728.693,E2 -4728.693} C_VEL
LIN {X 0,Y 523.916,Z 192.539,A -85,B 0,C 180,E1 -4731.08,E2 -4731.08} C_VEL
LIN {X 0,Y 523.895,Z 192.536,A -85,B 0,C 180,E1 -4733.824,E2 -4733.824} C_VEL
LIN {X 0,Y 523.942,Z 192.535,A -85,B 0,C 180,E1 -4736.635,E2 -4736.635} C_VEL
LIN {X 0,Y 523.949,Z 192.637,A -85,B 0,C 180,E1 -4739.856,E2 -4739.856} C_VEL
LIN {X 0,Y 528.741,Z 208.898,A -85,B 0,C 180,E1 -4741.736,E2 -4741.736} C_VEL
LIN {X 0,Y 528.819,Z 214.457,A -85,B 0,C 180,E1 -4742.279,E2 -4742.279} C_VEL
LIN {X 0,Y 528.151,Z 233.67,A -85,B 0,C 180,E1 -4744.086,E2 -4744.086} C_VEL
LIN {X 0,Y 530.886,Z 249.455,A -85,B 0,C 180,E1 -4744.465,E2 -4744.465} C_VEL
LIN {X 0,Y 529.307,Z 440.467,A -85,B 0,C 180,E1 -4747.197,E2 -4747.197} C_VEL
LIN {X 0,Y 528.968,Z 456.56,A -85,B 0,C 180,E1 -4747.568,E2 -4747.568} C_VEL
LIN {X 0,Y 528.513,Z 472.646,A -85,B 0,C 180,E1 -4748.088,E2 -4748.088} C_VEL
LIN {X 0,Y 528.018,Z 487.391,A -85,B 0,C 180,E1 -4748.702,E2 -4748.702} C_VEL
LIN {X 0,Y 527.357,Z 503.04,A -85,B 0,C 180,E1 -4749.522,E2 -4749.522} C_VEL
LIN {X 0,Y 526.795,Z 516.981,A -85,B 0,C 180,E1 -4750.415,E2 -4750.415} C_VEL
LIN {X 0,Y 526.157,Z 531.351,A -85,B 0,C 180,E1 -4751.506,E2 -4751.506} C_VEL
LIN {X 0,Y 525.568,Z 544.52,A -85,B 0,C 180,E1 -4752.689,E2 -4752.689} C_VEL
LIN {X 0,Y 525.079,Z 555.795,A -85,B 0,C 180,E1 -4753.874,E2 -4753.874} C_VEL
LIN {X 0,Y 524.617,Z 567.046,A -85,B 0,C 180,E1 -4755.253,E2 -4755.253} C_VEL
LIN {X 0,Y 524.178,Z 577.944,A -85,B 0,C 180,E1 -4756.823,E2 -4756.823} C_VEL
LIN {X 0,Y 523.936,Z 587.105,A -85,B 0,C 180,E1 -4758.391,E2 -4758.391} C_VEL
LIN {X 0,Y 523.659,Z 594.772,A -85,B 0,C 180,E1 -4759.951,E2 -4759.951} C_VEL
LIN {X 0,Y 523.505,Z 602.458,A -85,B 0,C 180,E1 -4761.895,E2 -4761.895} C_VEL
LIN {X 0,Y 523.412,Z 608.246,A -85,B 0,C 180,E1 -4763.832,E2 -4763.832} C_VEL
LIN {X 0,Y 523.312,Z 611.63,A -85,B 0,C 180,E1 -4765.376,E2 -4765.376} C_VEL
